LIN {X 0,Y 278.878,Z 465.633,A -85,B 0,C 180,E1 8845.226,E2 8845.226} C_VEL
LIN {X 0,Y 273.338,Z 453.94,A -85,B 0,C 180,E1 8842.303,E2 8842.303} C_VEL
LIN {X 0,Y 267.946,Z 443.512,A -85,B 0,C 180,E1 8839.057,E2 8839.057} C_VEL
LIN {X 0,Y 262.361,Z 433.364,A -85,B 0,C 180,E1 8835.019,E2 8835.019} C_VEL
LIN {X 0,Y 258.426,Z 426.882,A -85,B 0,C 180,E1 8831.493,E2 8831.493} C_VEL
LIN {X 0,Y 256.433,Z 423.717,A -85,B 0,C 180,E1 8829.312,E2 8829.312} C_VEL
LIN {X 0,Y 254.428,Z 420.112,A -85,B 0,C 180,E1 8826.543,E2 8826.543} C_VEL
LIN {X 0,Y 252.019,Z 415.913,A -85,B 0,C 180,E1 8821.364,E2 8821.364} C_VEL
LIN {X 0,Y 251.317,Z 414.93,A -85,B 0,C 180,E1 8815.664,E2 8815.664} C_VEL
LIN {X 0,Y 252.963,Z 416.019,A -85,B 0,C 180,E1 8809.754,E2 8809.754} C_VEL
LIN {X 0,Y 256.776,Z 421.342,A -85,B 0,C 180,E1 8803.95,E2 8803.95} C_VEL
LIN {X 0,Y 260.32,Z 426.562,A -85,B 0,C 180,E1 8800.361,E2 8800.361} C_VEL
LIN {X 0,Y 263.768,Z 431.814,A -85,B 0,C 180,E1 8797.547,E2 8797.547} C_VEL
LIN {X 0,Y 267.986,Z 438.368,A -85,B 0,C 180,E1 8794.65,E2 8794.65} C_VEL
LIN {X 0,Y 273.416,Z 447.764,A -85,B 0,C 180,E1 8791.435,E2 8791.435} C_VEL
LIN {X 0,Y 278.64,Z 457.79,A -85,B 0,C 180,E1 8788.724,E2 8788.724} C_VEL
LIN {X 0,Y 269.524,Z 577.471,A -85,B 0,C 180,E1 8786.054,E2 8786.054} C_VEL
LIN {X 0,Y 267.466,Z 596.812,A -85,B 0,C 180,E1 8785.36,E2 8785.36} C_VEL
LIN {X 0,Y 264.312,Z 615.233,A -85,B 0,C 180,E1 8784.419,E2 8784.419} C_VEL
LIN {X 0,Y 259.903,Z 633.791,A -85,B 0,C 180,E1 8783.145,E2 8783.145} C_VEL
LIN {X 0,Y 254.582,Z 651.308,A -85,B 0,C 180,E1 8781.583,E2 8781.583} C_VEL
LIN {X 0,Y 248.111,Z 668.635,A -85,B 0,C 180,E1 8779.608,E2 8779.608} C_VEL
LIN {X 0,Y 240.971,Z 684.785,A -85,B 0,C 180,E1 8777.257,E2 8777.257} C_VEL
LIN {X 0,Y 233.585,Z 699.288,A -85,B 0,C 180,E1 8774.586,E2 8774.586} C_VEL
LIN {X 0,Y 225.6,Z 713.172,A -85,B 0,C 180,E1 8771.327,E2 8771.327} C_VEL
LIN {X 0,Y 217.777,Z 725.421,A -85,B 0,C 180,E1 8767.634,E2 8767.634} C_VEL
LIN {X 0,Y 210.347,Z 736.116,A -85,B 0,C 180,E1 8763.461,E2 8763.461} C_VEL
LIN {X 0,Y 203.591,Z 745.264,A -85,B 0,C 180,E1 8758.769,E2 8758.769} C_VEL
LIN {X 0,Y 197.74,Z 752.844,A -85,B 0,C 180,E1 8753.544,E2 8753.544} C_VEL
LIN {X 0,Y 193.295,Z 758.557,A -85,B 0,C 180,E1 8748.081,E2 8748.081} C_VEL
LIN {X 0,Y 190.101,Z 762.723,A -85,B 0,C 180,E1 8742.145,E2 8742.145} C_VEL
LIN {X 0,Y 188.303,Z 765.165,A -85,B 0,C 180,E1 8736.096,E2 8736.096} C_VEL
LIN {X 0,Y 187.747,Z 765.976,A -85,B 0,C 180,E1 8730,E2 8730} C_VEL
LIN {X 0,Y 188.29,Z 765.2,A -85,B 0,C 180,E1 8723.904,E2 8723.904} C_VEL
LIN {X 0,Y 190.069,Z 762.799,A -85,B 0,C 180,E1 8717.853,E2 8717.853} C_VEL
LIN {X 0,Y 193.245,Z 758.673,A -85,B 0,C 180,E1 8711.915,E2 8711.915} C_VEL
LIN {X 0,Y 197.948,Z 752.674,A -85,B 0,C 180,E1 8706.167,E2 8706.167} C_VEL
LIN {X 0,Y 203.857,Z 745.036,A -85,B 0,C 180,E1 8700.951,E2 8700.951} C_VEL
LIN {X 0,Y 210.664,Z 735.828,A -85,B 0,C 180,E1 8696.269,E2 8696.269} C_VEL
LIN {X 0,Y 218.141,Z 725.064,A -85,B 0,C 180,E1 8692.108,E2 8692.108} C_VEL
LIN {X 0,Y 226.001,Z 712.736,A -85,B 0,C 180,E1 8688.425,E2 8688.425} C_VEL
LIN {X 0,Y 234.026,Z 698.729,A -85,B 0,C 180,E1 8685.172,E2 8685.172} C_VEL
LIN {X 0,Y 241.439,Z 684.148,A -85,B 0,C 180,E1 8682.513,E2 8682.513} C_VEL
LIN {X 0,Y 248.603,Z 667.849,A -85,B 0,C 180,E1 8680.17,E2 8680.17} C_VEL
LIN {X 0,Y 255.089,Z 650.314,A -85,B 0,C 180,E1 8678.199,E2 8678.199} C_VEL
LIN {X 0,Y 260.429,Z 632.572,A -85,B 0,C 180,E1 8676.641,E2 8676.641} C_VEL
LIN {X 0,Y 264.883,Z 613.37,A -85,B 0,C 180,E1 8675.356,E2 8675.356} C_VEL
LIN {X 0,Y 268.08,Z 593.774,A -85,B 0,C 180,E1 8674.394,E2 8674.394} C_VEL
LIN {X 0,Y 270.011,Z 573.44,A -85,B 0,C 180,E1 8673.717,E2 8673.717} C_VEL
LIN {X 0,Y 278.808,Z 457.69,A -85,B 0,C 180,E1 8671.152,E2 8671.152} C_VEL
LIN {X 0,Y 272.497,Z 445.95,A -85,B 0,C 180,E1 8667.839,E2 8667.839} C_VEL
LIN {X 0,Y 267.272,Z 437.11,A -85,B 0,C 180,E1 8664.653,E2 8664.653} C_VEL
LIN {X 0,Y 262.532,Z 429.641,A -85,B 0,C 180,E1 8661.212,E2 8661.212} C_VEL
LIN {X 0,Y 259.127,Z 424.746,A -85,B 0,C 180,E1 8658.213,E2 8658.213} C_VEL
LIN {X 0,Y 256.354,Z 420.667,A -85,B 0,C 180,E1 8655.149,E2 8655.149} C_VEL
LIN {X 0,Y 253.062,Z 416.095,A -85,B 0,C 180,E1 8649.782,E2 8649.782} C_VEL
LIN {X 0,Y 251.573,Z 415.164,A -85,B 0,C 180,E1 8643.875,E2 8643.875} C_VEL
LIN {X 0,Y 252.355,Z 416.185,A -85,B 0,C 180,E1 8638.411,E2 8638.411} C_VEL
LIN {X 0,Y 255.115,Z 421.076,A -85,B 0,C 180,E1 8632.796,E2 8632.796} C_VEL
LIN {X 0,Y 258.442,Z 426.742,A -85,B 0,C 180,E1 8628.734,E2 8628.734} C_VEL
LIN {X 0,Y 261.024,Z 431.187,A -85,B 0,C 180,E1 8626.272,E2 8626.272} C_VEL
LIN {X 0,Y 262.586,Z 435.115,A -85,B 0,C 180,E1 8624.85,E2 8624.85} C_VEL
LIN {X 0,Y 264.574,Z 443.488,A -85,B 0,C 180,E1 8622.933,E2 8622.933} C_VEL
LIN {X 0,Y 266.814,Z 452.064,A -85,B 0,C 180,E1 8621.05,E2 8621.05} C_VEL
LIN {X 0,Y 267.623,Z 454.063,A -85,B 0,C 180,E1 8620.49,E2 8620.49} C_VEL
LIN {X 0,Y 272.716,Z 464.616,A -85,B 0,C 180,E1 8617.416,E2 8617.416} C_VEL
LIN {X 0,Y 274.98,Z 470.078,A -85,B 0,C 180,E1 8616.14,E2 8616.14} C_VEL
LIN {X 0,Y 262.311,Z 614.422,A -85,B 0,C 180,E1 8612.779,E2 8612.779} C_VEL
LIN {X 0,Y 258.795,Z 635.834,A -85,B 0,C 180,E1 8612.035,E2 8612.035} C_VEL
LIN {X 0,Y 253.894,Z 656.209,A -85,B 0,C 180,E1 8611.07,E2 8611.07} C_VEL
LIN {X 0,Y 247.581,Z 676.274,A -85,B 0,C 180,E1 8609.793,E2 8609.793} C_VEL
LIN {X 0,Y 240.198,Z 695.651,A -85,B 0,C 180,E1 8608.12,E2 8608.12} C_VEL
LIN {X 0,Y 232.104,Z 713.934,A -85,B 0,C 180,E1 8606.019,E2 8606.019} C_VEL
LIN {X 0,Y 223.481,Z 731.176,A -85,B 0,C 180,E1 8603.423,E2 8603.423} C_VEL
LIN {X 0,Y 214.547,Z 747.362,A -85,B 0,C 180,E1 8600.258,E2 8600.258} C_VEL
LIN {X 0,Y 205.621,Z 762.427,A -85,B 0,C 180,E1 8596.428,E2 8596.428} C_VEL
LIN {X 0,Y 197.354,Z 775.9,A -85,B 0,C 180,E1 8591.969,E2 8591.969} C_VEL
LIN {X 0,Y 190.055,Z 787.822,A -85,B 0,C 180,E1 8586.85,E2 8586.85} C_VEL
LIN {X 0,Y 184.137,Z 798.176,A -85,B 0,C 180,E1 8581.053,E2 8581.053} C_VEL
LIN {X 0,Y 180.13,Z 806.495,A -85,B 0,C 180,E1 8574.951,E2 8574.951} C_VEL
LIN {X 0,Y 177.989,Z 812.955,A -85,B 0,C 180,E1 8568.674,E2 8568.674} C_VEL
LIN {X 0,Y 177.55,Z 817.657,A -85,B 0,C 180,E1 8562.356,E2 8562.356} C_VEL
LIN {X 0,Y 178.282,Z 820.523,A -85,B 0,C 180,E1 8556.44,E2 8556.44} C_VEL
LIN {X 0,Y 179.036,Z 821.548,A -85,B 0,C 180,E1 8551.92,E2 8551.92} C_VEL
LIN {X 0,Y 179.07,Z 821.577,A -85,B 0,C 180,E1 8548.4,E2 8548.4} C_VEL
LIN {X 0,Y 178.404,Z 820.702,A -85,B 0,C 180,E1 8544.21,E2 8544.21} C_VEL
LIN {X 0,Y 177.589,Z 818.027,A -85,B 0,C 180,E1 8538.306,E2 8538.306} C_VEL
LIN {X 0,Y 177.869,Z 813.516,A -85,B 0,C 180,E1 8531.991,E2 8531.991} C_VEL
LIN {X 0,Y 179.816,Z 807.245,A -85,B 0,C 180,E1 8525.703,E2 8525.703} C_VEL
LIN {X 0,Y 183.877,Z 798.609,A -85,B 0,C 180,E1 8519.261,E2 8519.261} C_VEL
LIN {X 0,Y 189.692,Z 788.341,A -85,B 0,C 180,E1 8513.445,E2 8513.445} C_VEL
LIN {X 0,Y 196.965,Z 776.407,A -85,B 0,C 180,E1 8508.263,E2 8508.263} C_VEL
LIN {X 0,Y 205.148,Z 763.047,A -85,B 0,C 180,E1 8503.795,E2 8503.795} C_VEL
LIN {X 0,Y 213.949,Z 748.192,A -85,B 0,C 180,E1 8499.968,E2 8499.968} C_VEL
LIN {X 0,Y 222.83,Z 732.143,A -85,B 0,C 180,E1 8496.782,E2 8496.782} C_VEL
LIN {X 0,Y 231.368,Z 715.151,A -85,B 0,C 180,E1 8494.18,E2 8494.18} C_VEL
LIN {X 0,Y 239.105,Z 697.83,A -85,B 0,C 180,E1 8492.138,E2 8492.138} C_VEL
LIN {X 0,Y 246.063,Z 679.96,A -85,B 0,C 180,E1 8490.524,E2 8490.524} C_VEL
LIN {X 0,Y 252.141,Z 661.532,A -85,B 0,C 180,E1 8489.264,E2 8489.264} C_VEL
LIN {X 0,Y 257.488,Z 640.986,A -85,B 0,C 180,E1 8488.212,E2 8488.212} C_VEL
LIN {X 0,Y 261.349,Z 619.931,A -85,B 0,C 180,E1 8487.418,E2 8487.418} C_VEL
LIN {X 0,Y 264.036,Z 594.652,A -85,B 0,C 180,E1 8486.746,E2 8486.746} C_VEL
LIN {X 0,Y 274.757,Z 469.441,A -85,B 0,C 180,E1 8483.824,E2 8483.824} C_VEL
LIN {X 0,Y 269.41,Z 457.799,A -85,B 0,C 180,E1 8480.758,E2 8480.758} C_VEL
LIN {X 0,Y 263.947,Z 447.113,A -85,B 0,C 180,E1 8477.129,E2 8477.129} C_VEL
LIN {X 0,Y 259.778,Z 439.543,A -85,B 0,C 180,E1 8473.805,E2 8473.805} C_VEL
LIN {X 0,Y 256.77,Z 434.226,A -85,B 0,C 180,E1 8470.886,E2 8470.886} C_VEL
LIN {X 0,Y 253.434,Z 428.163,A -85,B 0,C 180,E1 8466.569,E2 8466.569} C_VEL
LIN {X 0,Y 250.96,Z 423.8,A -85,B 0,C 180,E1 8461.141,E2 8461.141} C_VEL
LIN {X 0,Y 250.345,Z 422.871,A -85,B 0,C 180,E1 8455.647,E2 8455.647} C_VEL
LIN {X 0,Y 252.001,Z 423.991,A -85,B 0,C 180,E1 8449.714,E2 8449.714} C_VEL
LIN {X 0,Y 255.526,Z 429.237,A -85,B 0,C 180,E1 8444.219,E2 8444.219} C_VEL
LIN {X 0,Y 258.761,Z 434.142,A -85,B 0,C 180,E1 8440.825,E2 8440.825} C_VEL
LIN {X 0,Y 262.133,Z 439.449,A -85,B 0,C 180,E1 8437.971,E2 8437.971} C_VEL
LIN {X 0,Y 266.367,Z 446.383,A -85,B 0,C 180,E1 8434.961,E2 8434.961} C_VEL
LIN {X 0,Y 271.172,Z 455.032,A -85,B 0,C 180,E1 8432.017,E2 8432.017} C_VEL
LIN {X 0,Y 274.625,Z 461.918,A -85,B 0,C 180,E1 8430.11,E2 8430.11} C_VEL
LIN {X 0,Y 265.44,Z 578.24,A -85,B 0,C 180,E1 8427.518,E2 8427.518} C_VEL
LIN {X 0,Y 263.304,Z 597.581,A -85,B 0,C 180,E1 8426.825,E2 8426.825} C_VEL
LIN {X 0,Y 260.034,Z 616.06,A -85,B 0,C 180,E1 8425.886,E2 8425.886} C_VEL
LIN {X 0,Y 255.561,Z 634.361,A -85,B 0,C 180,E1 8424.639,E2 8424.639} C_VEL
LIN {X 0,Y 250.09,Z 651.862,A -85,B 0,C 180,E1 8423.09,E2 8423.09} C_VEL
LIN {X 0,Y 243.394,Z 669.282,A -85,B 0,C 180,E1 8421.118,E2 8421.118} C_VEL
LIN {X 0,Y 235.981,Z 685.526,A -85,B 0,C 180,E1 8418.762,E2 8418.762} C_VEL
LIN {X 0,Y 228.025,Z 700.565,A -85,B 0,C 180,E1 8415.98,E2 8415.98} C_VEL
LIN {X 0,Y 219.721,Z 714.42,A -85,B 0,C 180,E1 8412.689,E2 8412.689} C_VEL
LIN {X 0,Y 211.561,Z 726.652,A -85,B 0,C 180,E1 8408.944,E2 8408.944} C_VEL
LIN {X 0,Y 203.781,Z 737.336,A -85,B 0,C 180,E1 8404.69,E2 8404.69} C_VEL
LIN {X 0,Y 196.675,Z 746.477,A -85,B 0,C 180,E1 8399.881,E2 8399.881} C_VEL
LIN {X 0,Y 190.493,Z 754.053,A -85,B 0,C 180,E1 8394.497,E2 8394.497} C_VEL
LIN {X 0,Y 185.77,Z 759.763,A -85,B 0,C 180,E1 8388.84,E2 8388.84} C_VEL
LIN {X 0,Y 182.363,Z 763.927,A -85,B 0,C 180,E1 8382.668,E2 8382.668} C_VEL
LIN {X 0,Y 180.435,Z 766.367,A -85,B 0,C 180,E1 8376.363,E2 8376.363} C_VEL
LIN {X 0,Y 179.838,Z 767.178,A -85,B 0,C 180,E1 8370,E2 8370} C_VEL
LIN {X 0,Y 180.422,Z 766.402,A -85,B 0,C 180,E1 8363.637,E2 8363.637} C_VEL
LIN {X 0,Y 182.33,Z 764.002,A -85,B 0,C 180,E1 8357.329,E2 8357.329} C_VEL
LIN {X 0,Y 185.719,Z 759.877,A -85,B 0,C 180,E1 8351.155,E2 8351.155} C_VEL
LIN {X 0,Y 190.717,Z 753.881,A -85,B 0,C 180,E1 8345.203,E2 8345.203} C_VEL
LIN {X 0,Y 196.958,Z 746.25,A -85,B 0,C 180,E1 8339.831,E2 8339.831} C_VEL
LIN {X 0,Y 204.119,Z 737.048,A -85,B 0,C 180,E1 8335.034,E2 8335.034} C_VEL
LIN {X 0,Y 211.947,Z 726.296,A -85,B 0,C 180,E1 8330.793,E2 8330.793} C_VEL
LIN {X 0,Y 220.146,Z 713.986,A -85,B 0,C 180,E1 8327.059,E2 8327.059} C_VEL
LIN {X 0,Y 228.485,Z 700.025,A -85,B 0,C 180,E1 8323.778,E2 8323.778} C_VEL
LIN {X 0,Y 236.481,Z 684.837,A -85,B 0,C 180,E1 8321.002,E2 8321.002} C_VEL
LIN {X 0,Y 243.906,Z 668.454,A -85,B 0,C 180,E1 8318.657,E2 8318.657} C_VEL
LIN {X 0,Y 250.266,Z 651.876,A -85,B 0,C 180,E1 8316.793,E2 8316.793} C_VEL
LIN {X 0,Y 255.814,Z 634.148,A -85,B 0,C 180,E1 8315.228,E2 8315.228} C_VEL
LIN {X 0,Y 260.374,Z 615.388,A -85,B 0,C 180,E1 8313.96,E2 8313.96} C_VEL
LIN {X 0,Y 263.777,Z 595.743,A -85,B 0,C 180,E1 8312.979,E2 8312.979} C_VEL
LIN {X 0,Y 265.852,Z 575.618,A -85,B 0,C 180,E1 8312.291,E2 8312.291} C_VEL
LIN {X 0,Y 274.724,Z 461.747,A -85,B 0,C 180,E1 8309.729,E2 8309.729} C_VEL
LIN {X 0,Y 269.186,Z 451.135,A -85,B 0,C 180,E1 8306.589,E2 8306.589} C_VEL
LIN {X 0,Y 264.409,Z 442.959,A -85,B 0,C 180,E1 8303.454,E2 8303.454} C_VEL
LIN {X 0,Y 260.148,Z 436.17,A -85,B 0,C 180,E1 8300.12,E2 8300.12} C_VEL
LIN {X 0,Y 257.621,Z 432.313,A -85,B 0,C 180,E1 8297.739,E2 8297.739} C_VEL
LIN {X 0,Y 255.045,Z 428.396,A -85,B 0,C 180,E1 8294.763,E2 8294.763} C_VEL
LIN {X 0,Y 252.008,Z 423.989,A -85,B 0,C 180,E1 8289.593,E2 8289.593} C_VEL
LIN {X 0,Y 250.592,Z 423.106,A -85,B 0,C 180,E1 8283.661,E2 8283.661} C_VEL
LIN {X 0,Y 251.362,Z 424.279,A -85,B 0,C 180,E1 8278.405,E2 8278.405} C_VEL
LIN {X 0,Y 253.873,Z 428.918,A -85,B 0,C 180,E1 8273.101,E2 8273.101} C_VEL
LIN {X 0,Y 256.901,Z 434.265,A -85,B 0,C 180,E1 8269.233,E2 8269.233} C_VEL
LIN {X 0,Y 260.684,Z 440.814,A -85,B 0,C 180,E1 8265.621,E2 8265.621} C_VEL
LIN {X 0,Y 265.967,Z 450.804,A -85,B 0,C 180,E1 8261.592,E2 8261.592} C_VEL
LIN {X 0,Y 267.623,Z 454.063,A -85,B 0,C 180,E1 8260.49,E2 8260.49} C_VEL
LIN {X 0,Y 268.653,Z 457.702,A -85,B 0,C 180,E1 8259.728,E2 8259.728} C_VEL
LIN {X 0,Y 270.267,Z 470.787,A -85,B 0,C 180,E1 8258.119,E2 8258.119} C_VEL
LIN {X 0,Y 271.051,Z 473.538,A -85,B 0,C 180,E1 8257.597,E2 8257.597} C_VEL
LIN {X 0,Y 258.457,Z 613.492,A -85,B 0,C 180,E1 8254.336,E2 8254.336} C_VEL
LIN {X 0,Y 254.871,Z 634.831,A -85,B 0,C 180,E1 8253.607,E2 8253.607} C_VEL
LIN {X 0,Y 249.872,Z 655.168,A -85,B 0,C 180,E1 8252.661,E2 8252.661} C_VEL
LIN {X 0,Y 243.592,Z 674.701,A -85,B 0,C 180,E1 8251.446,E2 8251.446} C_VEL
LIN {X 0,Y 235.986,Z 694.185,A -85,B 0,C 180,E1 8249.804,E2 8249.804} C_VEL
LIN {X 0,Y 227.614,Z 712.526,A -85,B 0,C 180,E1 8247.735,E2 8247.735} C_VEL
LIN {X 0,Y 218.527,Z 730.074,A -85,B 0,C 180,E1 8245.116,E2 8245.116} C_VEL
LIN {X 0,Y 209.154,Z 746.368,A -85,B 0,C 180,E1 8241.926,E2 8241.926} C_VEL
LIN {X 0,Y 199.978,Z 761.113,A -85,B 0,C 180,E1 8238.155,E2 8238.155} C_VEL
LIN {X 0,Y 191.242,Z 774.603,A -85,B 0,C 180,E1 8233.639,E2 8233.639} C_VEL
LIN {X 0,Y 183.44,Z 786.534,A -85,B 0,C 180,E1 8228.415,E2 8228.415} C_VEL
LIN {X 0,Y 177.041,Z 796.897,A -85,B 0,C 180,E1 8222.446,E2 8222.446} C_VEL
LIN {X 0,Y 172.62,Z 805.225,A -85,B 0,C 180,E1 8216.116,E2 8216.116} C_VEL
LIN {X 0,Y 170.181,Z 811.698,A -85,B 0,C 180,E1 8209.565,E2 8209.565} C_VEL
LIN {X 0,Y 169.577,Z 816.415,A -85,B 0,C 180,E1 8202.947,E2 8202.947} C_VEL
LIN {X 0,Y 170.287,Z 819.301,A -85,B 0,C 180,E1 8196.744,E2 8196.744} C_VEL
LIN {X 0,Y 171.107,Z 820.343,A -85,B 0,C 180,E1 8192.009,E2 8192.009} C_VEL
LIN {X 0,Y 171.178,Z 820.405,A -85,B 0,C 180,E1 8188.661,E2 8188.661} C_VEL
LIN {X 0,Y 170.476,Z 819.577,A -85,B 0,C 180,E1 8184.278,E2 8184.278} C_VEL
LIN {X 0,Y 169.621,Z 816.985,A -85,B 0,C 180,E1 8178.094,E2 8178.094} C_VEL
LIN {X 0,Y 169.97,Z 812.559,A -85,B 0,C 180,E1 8171.479,E2 8171.479} C_VEL
LIN {X 0,Y 172.273,Z 805.975,A -85,B 0,C 180,E1 8164.566,E2 8164.566} C_VEL
LIN {X 0,Y 176.757,Z 797.329,A -85,B 0,C 180,E1 8157.879,E2 8157.879} C_VEL
LIN {X 0,Y 183.113,Z 786.955,A -85,B 0,C 180,E1 8151.839,E2 8151.839} C_VEL
LIN {X 0,Y 190.759,Z 775.213,A -85,B 0,C 180,E1 8146.637,E2 8146.637} C_VEL
LIN {X 0,Y 199.421,Z 761.827,A -85,B 0,C 180,E1 8142.096,E2 8142.096} C_VEL
LIN {X 0,Y 208.727,Z 746.868,A -85,B 0,C 180,E1 8138.225,E2 8138.225} C_VEL
LIN {X 0,Y 217.99,Z 730.79,A -85,B 0,C 180,E1 8135.045,E2 8135.045} C_VEL
LIN {X 0,Y 226.895,Z 713.67,A -85,B 0,C 180,E1 8132.45,E2 8132.45} C_VEL
LIN {X 0,Y 235.227,Z 695.538,A -85,B 0,C 180,E1 8130.362,E2 8130.362} C_VEL
LIN {X 0,Y 242.416,Z 677.385,A -85,B 0,C 180,E1 8128.784,E2 8128.784} C_VEL
LIN {X 0,Y 248.711,Z 658.403,A -85,B 0,C 180,E1 8127.548,E2 8127.548} C_VEL
LIN {X 0,Y 253.921,Z 638.253,A -85,B 0,C 180,E1 8126.563,E2 8126.563} C_VEL
LIN {X 0,Y 257.673,Z 617.588,A -85,B 0,C 180,E1 8125.814,E2 8125.814} C_VEL
LIN {X 0,Y 260.622,Z 589.211,A -85,B 0,C 180,E1 8125.086,E2 8125.086} C_VEL
LIN {X 0,Y 270.847,Z 473.338,A -85,B 0,C 180,E1 8122.405,E2 8122.405} C_VEL
LIN {X 0,Y 266.038,Z 462.77,A -85,B 0,C 180,E1 8119.427,E2 8119.427} C_VEL
LIN {X 0,Y 261.467,Z 453.484,A -85,B 0,C 180,E1 8116.152,E2 8116.152} C_VEL
LIN {X 0,Y 257.896,Z 446.68,A -85,B 0,C 180,E1 8113.109,E2 8113.109} C_VEL
LIN {X 0,Y 254.958,Z 441.205,A -85,B 0,C 180,E1 8110.05,E2 8110.05} C_VEL
LIN {X 0,Y 251.865,Z 435.512,A -85,B 0,C 180,E1 8105.695,E2 8105.695} C_VEL
LIN {X 0,Y 249.905,Z 431.687,A -85,B 0,C 180,E1 8100.917,E2 8100.917} C_VEL
LIN {X 0,Y 249.389,Z 430.818,A -85,B 0,C 180,E1 8095.4,E2 8095.4} C_VEL
LIN {X 0,Y 250.937,Z 431.891,A -85,B 0,C 180,E1 8089.902,E2 8089.902} C_VEL
LIN {X 0,Y 254.192,Z 436.961,A -85,B 0,C 180,E1 8084.602,E2 8084.602} C_VEL
LIN {X 0,Y 257.218,Z 441.719,A -85,B 0,C 180,E1 8081.295,E2 8081.295} C_VEL
LIN {X 0,Y 260.737,Z 447.429,A -85,B 0,C 180,E1 8078.221,E2 8078.221} C_VEL
LIN {X 0,Y 265.223,Z 455.175,A -85,B 0,C 180,E1 8074.965,E2 8074.965} C_VEL
LIN {X 0,Y 270.149,Z 464.689,A -85,B 0,C 180,E1 8071.902,E2 8071.902} C_VEL
LIN {X 0,Y 270.764,Z 466.184,A -85,B 0,C 180,E1 8071.534,E2 8071.534} C_VEL
LIN {X 0,Y 261.543,Z 578.894,A -85,B 0,C 180,E1 8069.031,E2 8069.031} C_VEL
LIN {X 0,Y 259.335,Z 598.253,A -85,B 0,C 180,E1 8068.341,E2 8068.341} C_VEL
LIN {X 0,Y 256.033,Z 616.456,A -85,B 0,C 180,E1 8067.426,E2 8067.426} C_VEL
LIN {X 0,Y 251.465,Z 634.7,A -85,B 0,C 180,E1 8066.2,E2 8066.2} C_VEL
LIN {X 0,Y 245.442,Z 653.314,A -85,B 0,C 180,E1 8064.559,E2 8064.559} C_VEL
LIN {X 0,Y 238.524,Z 670.647,A -85,B 0,C 180,E1 8062.592,E2 8062.592} C_VEL
LIN {X 0,Y 230.865,Z 686.815,A -85,B 0,C 180,E1 8060.239,E2 8060.239} C_VEL
LIN {X 0,Y 222.606,Z 701.837,A -85,B 0,C 180,E1 8057.443,E2 8057.443} C_VEL
LIN {X 0,Y 213.973,Z 715.667,A -85,B 0,C 180,E1 8054.125,E2 8054.125} C_VEL
LIN {X 0,Y 205.461,Z 727.883,A -85,B 0,C 180,E1 8050.332,E2 8050.332} C_VEL
LIN {X 0,Y 197.315,Z 738.556,A -85,B 0,C 180,E1 8046.001,E2 8046.001} C_VEL
LIN {X 0,Y 189.838,Z 747.69,A -85,B 0,C 180,E1 8041.074,E2 8041.074} C_VEL
LIN {X 0,Y 183.302,Z 755.261,A -85,B 0,C 180,E1 8035.525,E2 8035.525} C_VEL
LIN {X 0,Y 178.101,Z 761.156,A -85,B 0,C 180,E1 8029.41,E2 8029.41} C_VEL
LIN {X 0,Y 174.64,Z 765.131,A -85,B 0,C 180,E1 8023.239,E2 8023.239} C_VEL
LIN {X 0,Y 172.572,Z 767.569,A -85,B 0,C 180,E1 8016.654,E2 8016.654} C_VEL
LIN {X 0,Y 171.929,Z 768.379,A -85,B 0,C 180,E1 8010,E2 8010} C_VEL
LIN {X 0,Y 172.558,Z 767.603,A -85,B 0,C 180,E1 8003.345,E2 8003.345} C_VEL
LIN {X 0,Y 174.606,Z 765.204,A -85,B 0,C 180,E1 7996.759,E2 7996.759} C_VEL
LIN {X 0,Y 178.23,Z 761.081,A -85,B 0,C 180,E1 7990.331,E2 7990.331} C_VEL
LIN {X 0,Y 183.543,Z 755.089,A -85,B 0,C 180,E1 7984.165,E2 7984.165} C_VEL
LIN {X 0,Y 190.141,Z 747.462,A -85,B 0,C 180,E1 7978.629,E2 7978.629} C_VEL
LIN {X 0,Y 197.674,Z 738.268,A -85,B 0,C 180,E1 7973.716,E2 7973.716} C_VEL
LIN {X 0,Y 205.871,Z 727.526,A -85,B 0,C 180,E1 7969.4,E2 7969.4} C_VEL
LIN {X 0,Y 214.422,Z 715.233,A -85,B 0,C 180,E1 7965.618,E2 7965.618} C_VEL
LIN {X 0,Y 223.091,Z 701.302,A -85,B 0,C 180,E1 7962.313,E2 7962.313} C_VEL
LIN {X 0,Y 231.381,Z 686.158,A -85,B 0,C 180,E1 7959.527,E2 7959.527} C_VEL
LIN {X 0,Y 239.064,Z 669.839,A -85,B 0,C 180,E1 7957.182,E2 7957.182} C_VEL
LIN {X 0,Y 245.998,Z 652.299,A -85,B 0,C 180,E1 7955.22,E2 7955.22} C_VEL
LIN {X 0,Y 251.698,Z 634.574,A -85,B 0,C 180,E1 7953.674,E2 7953.674} C_VEL
LIN {X 0,Y 256.472,Z 615.362,A -85,B 0,C 180,E1 7952.396,E2 7952.396} C_VEL
LIN {X 0,Y 259.942,Z 595.562,A -85,B 0,C 180,E1 7951.429,E2 7951.429} C_VEL
LIN {X 0,Y 262.042,Z 575.24,A -85,B 0,C 180,E1 7950.751,E2 7950.751} C_VEL
LIN {X 0,Y 270.904,Z 465.97,A -85,B 0,C 180,E1 7948.313,E2 7948.313} C_VEL
LIN {X 0,Y 265.845,Z 456.132,A -85,B 0,C 180,E1 7945.211,E2 7945.211} C_VEL
LIN {X 0,Y 261.321,Z 448.177,A -85,B 0,C 180,E1 7941.964,E2 7941.964} C_VEL
LIN {X 0,Y 257.639,Z 442.271,A -85,B 0,C 180,E1 7938.791,E2 7938.791} C_VEL
LIN {X 0,Y 255.622,Z 439.169,A -85,B 0,C 180,E1 7936.708,E2 7936.708} C_VEL
LIN {X 0,Y 253.747,Z 436.123,A -85,B 0,C 180,E1 7934.374,E2 7934.374} C_VEL
LIN {X 0,Y 250.952,Z 431.883,A -85,B 0,C 180,E1 7929.402,E2 7929.402} C_VEL
LIN {X 0,Y 249.613,Z 431.063,A -85,B 0,C 180,E1 7923.445,E2 7923.445} C_VEL
LIN {X 0,Y 250.31,Z 432.173,A -85,B 0,C 180,E1 7918.627,E2 7918.627} C_VEL
LIN {X 0,Y 252.595,Z 436.657,A -85,B 0,C 180,E1 7913.482,E2 7913.482} C_VEL
LIN {X 0,Y 255.473,Z 441.965,A -85,B 0,C 180,E1 7909.629,E2 7909.629} C_VEL
LIN {X 0,Y 259.181,Z 448.801,A -85,B 0,C 180,E1 7905.934,E2 7905.934} C_VEL
LIN {X 0,Y 263.838,Z 457.95,A -85,B 0,C 180,E1 7902.238,E2 7902.238} C_VEL
LIN {X 0,Y 268.608,Z 468.029,A -85,B 0,C 180,E1 7899.063,E2 7899.063} C_VEL
LIN {X 0,Y 271.051,Z 473.538,A -85,B 0,C 180,E1 7897.597,E2 7897.597} C_VEL
LIN {X 0,Y 271.539,Z 476.413,A -85,B 0,C 180,E1 7897.208,E2 7897.208} C_VEL
LIN {X 0,Y 271.269,Z 480.92,A -85,B 0,C 180,E1 7897.051,E2 7897.051} C_VEL
LIN {X 0,Y 269.929,Z 487.325,A -85,B 0,C 180,E1 7897.239,E2 7897.239} C_VEL
LIN {X 0,Y 265.57,Z 502.194,A -85,B 0,C 180,E1 7898.257,E2 7898.257} C_VEL
LIN {X 0,Y 264.534,Z 508.324,A -85,B 0,C 180,E1 7898.34,E2 7898.34} C_VEL
LIN {X 0,Y 254.757,Z 612.84,A -85,B 0,C 180,E1 7895.931,E2 7895.931} C_VEL
LIN {X 0,Y 251.088,Z 634.078,A -85,B 0,C 180,E1 7895.216,E2 7895.216} C_VEL
LIN {X 0,Y 245.844,Z 654.788,A -85,B 0,C 180,E1 7894.266,E2 7894.266} C_VEL
LIN {X 0,Y 239.415,Z 674.224,A -85,B 0,C 180,E1 7893.075,E2 7893.075} C_VEL
LIN {X 0,Y 231.603,Z 693.598,A -85,B 0,C 180,E1 7891.463,E2 7891.463} C_VEL
LIN {X 0,Y 222.975,Z 711.859,A -85,B 0,C 180,E1 7889.422,E2 7889.422} C_VEL
LIN {X 0,Y 213.717,Z 729.073,A -85,B 0,C 180,E1 7886.868,E2 7886.868} C_VEL
LIN {X 0,Y 204.038,Z 745.225,A -85,B 0,C 180,E1 7883.715,E2 7883.715} C_VEL
LIN {X 0,Y 194.533,Z 759.801,A -85,B 0,C 180,E1 7879.979,E2 7879.979} C_VEL
LIN {X 0,Y 185.3,Z 773.305,A -85,B 0,C 180,E1 7875.417,E2 7875.417} C_VEL
LIN {X 0,Y 176.976,Z 785.247,A -85,B 0,C 180,E1 7870.094,E2 7870.094} C_VEL
LIN {X 0,Y 170.06,Z 795.62,A -85,B 0,C 180,E1 7863.954,E2 7863.954} C_VEL
LIN {X 0,Y 165.185,Z 803.954,A -85,B 0,C 180,E1 7857.388,E2 7857.388} C_VEL
LIN {X 0,Y 162.407,Z 810.439,A -85,B 0,C 180,E1 7850.543,E2 7850.543} C_VEL
LIN {X 0,Y 161.613,Z 815.173,A -85,B 0,C 180,E1 7843.597,E2 7843.597} C_VEL
LIN {X 0,Y 162.282,Z 818.076,A -85,B 0,C 180,E1 7837.078,E2 7837.078} C_VEL
LIN {X 0,Y 163.175,Z 819.137,A -85,B 0,C 180,E1 7832.107,E2 7832.107} C_VEL
LIN {X 0,Y 163.256,Z 819.202,A -85,B 0,C 180,E1 7828.596,E2 7828.596} C_VEL
LIN {X 0,Y 162.481,Z 818.356,A -85,B 0,C 180,E1 7823.995,E2 7823.995} C_VEL
LIN {X 0,Y 161.638,Z 815.742,A -85,B 0,C 180,E1 7817.497,E2 7817.497} C_VEL
LIN {X 0,Y 162.159,Z 811.3,A -85,B 0,C 180,E1 7810.552,E2 7810.552} C_VEL
LIN {X 0,Y 164.796,Z 804.703,A -85,B 0,C 180,E1 7803.323,E2 7803.323} C_VEL
LIN {X 0,Y 169.748,Z 796.048,A -85,B 0,C 180,E1 7796.381,E2 7796.381} C_VEL
LIN {X 0,Y 176.556,Z 785.763,A -85,B 0,C 180,E1 7790.215,E2 7790.215} C_VEL
LIN {X 0,Y 184.79,Z 773.917,A -85,B 0,C 180,E1 7784.863,E2 7784.863} C_VEL
LIN {X 0,Y 193.946,Z 760.519,A -85,B 0,C 180,E1 7780.273,E2 7780.273} C_VEL
LIN {X 0,Y 203.708,Z 745.539,A -85,B 0,C 180,E1 7776.396,E2 7776.396} C_VEL
LIN {X 0,Y 213.209,Z 729.692,A -85,B 0,C 180,E1 7773.276,E2 7773.276} C_VEL
LIN {X 0,Y 222.597,Z 712.279,A -85,B 0,C 180,E1 7770.666,E2 7770.666} C_VEL
LIN {X 0,Y 231.206,Z 694.085,A -85,B 0,C 180,E1 7768.615,E2 7768.615} C_VEL
LIN {X 0,Y 238.607,Z 675.837,A -85,B 0,C 180,E1 7767.072,E2 7767.072} C_VEL
LIN {X 0,Y 245.023,Z 656.831,A -85,B 0,C 180,E1 7765.873,E2 7765.873} C_VEL
LIN {X 0,Y 250.242,Z 636.931,A -85,B 0,C 180,E1 7764.927,E2 7764.927} C_VEL
LIN {X 0,Y 254.035,Z 616.367,A -85,B 0,C 180,E1 7764.2,E2 7764.2} C_VEL
LIN {X 0,Y 257.092,Z 587.514,A -85,B 0,C 180,E1 7763.472,E2 7763.472} C_VEL
LIN {X 0,Y 267.095,Z 477.349,A -85,B 0,C 180,E1 7760.946,E2 7760.946} C_VEL
LIN {X 0,Y 262.464,Z 466.849,A -85,B 0,C 180,E1 7757.801,E2 7757.801} C_VEL
LIN {X 0,Y 257.967,Z 457.509,A -85,B 0,C 180,E1 7754.19,E2 7754.19} C_VEL
LIN {X 0,Y 254.309,Z 450.317,A -85,B 0,C 180,E1 7750.534,E2 7750.534} C_VEL
LIN {X 0,Y 252.182,Z 446.451,A -85,B 0,C 180,E1 7747.861,E2 7747.861} C_VEL
LIN {X 0,Y 250.603,Z 443.213,A -85,B 0,C 180,E1 7745.265,E2 7745.265} C_VEL
LIN {X 0,Y 248.856,Z 439.575,A -85,B 0,C 180,E1 7740.69,E2 7740.69} C_VEL
LIN {X 0,Y 248.41,Z 438.758,A -85,B 0,C 180,E1 7735.382,E2 7735.382} C_VEL
LIN {X 0,Y 249.865,Z 439.829,A -85,B 0,C 180,E1 7730.091,E2 7730.091} C_VEL
LIN {X 0,Y 252.865,Z 444.683,A -85,B 0,C 180,E1 7724.989,E2 7724.989} C_VEL
LIN {X 0,Y 255.69,Z 449.295,A -85,B 0,C 180,E1 7721.769,E2 7721.769} C_VEL
LIN {X 0,Y 259.434,Z 455.525,A -85,B 0,C 180,E1 7718.404,E2 7718.404} C_VEL
LIN {X 0,Y 264.142,Z 464.247,A -85,B 0,C 180,E1 7714.915,E2 7714.915} C_VEL
LIN {X 0,Y 267.074,Z 470.47,A -85,B 0,C 180,E1 7712.997,E2 7712.997} C_VEL
LIN {X 0,Y 257.843,Z 579.44,A -85,B 0,C 180,E1 7710.592,E2 7710.592} C_VEL
LIN {X 0,Y 255.589,Z 598.711,A -85,B 0,C 180,E1 7709.912,E2 7709.912} C_VEL
LIN {X 0,Y 252.035,Z 617.628,A -85,B 0,C 180,E1 7708.968,E2 7708.968} C_VEL
LIN {X 0,Y 247.178,Z 636.274,A -85,B 0,C 180,E1 7707.715,E2 7707.715} C_VEL
LIN {X 0,Y 241.308,Z 653.871,A -85,B 0,C 180,E1 7706.175,E2 7706.175} C_VEL
LIN {X 0,Y 234.158,Z 671.292,A -85,B 0,C 180,E1 7704.221,E2 7704.221} C_VEL
LIN {X 0,Y 226.228,Z 687.532,A -85,B 0,C 180,E1 7701.877,E2 7701.877} C_VEL
LIN {X 0,Y 217.745,Z 702.468,A -85,B 0,C 180,E1 7699.116,E2 7699.116} C_VEL
LIN {X 0,Y 208.949,Z 716.095,A -85,B 0,C 180,E1 7695.869,E2 7695.869} C_VEL
LIN {X 0,Y 200.025,Z 728.437,A -85,B 0,C 180,E1 7692.052,E2 7692.052} C_VEL
LIN {X 0,Y 191.434,Z 739.221,A -85,B 0,C 180,E1 7687.667,E2 7687.667} C_VEL
LIN {X 0,Y 183.495,Z 748.46,A -85,B 0,C 180,E1 7682.645,E2 7682.645} C_VEL
LIN {X 0,Y 176.504,Z 756.135,A -85,B 0,C 180,E1 7676.947,E2 7676.947} C_VEL
LIN {X 0,Y 170.775,Z 762.231,A -85,B 0,C 180,E1 7670.481,E2 7670.481} C_VEL
LIN {X 0,Y 166.936,Z 766.334,A -85,B 0,C 180,E1 7663.861,E2 7663.861} C_VEL
LIN {X 0,Y 164.713,Z 768.772,A -85,B 0,C 180,E1 7656.973,E2 7656.973} C_VEL
LIN {X 0,Y 164.019,Z 769.581,A -85,B 0,C 180,E1 7650,E2 7650} C_VEL
LIN {X 0,Y 164.698,Z 768.805,A -85,B 0,C 180,E1 7643.026,E2 7643.026} C_VEL
LIN {X 0,Y 167.009,Z 766.307,A -85,B 0,C 180,E1 7635.902,E2 7635.902} C_VEL
LIN {X 0,Y 171.022,Z 762.045,A -85,B 0,C 180,E1 7629.107,E2 7629.107} C_VEL
LIN {X 0,Y 176.764,Z 755.939,A -85,B 0,C 180,E1 7622.732,E2 7622.732} C_VEL
LIN {X 0,Y 183.818,Z 748.206,A -85,B 0,C 180,E1 7617.049,E2 7617.049} C_VEL
LIN {X 0,Y 191.816,Z 738.903,A -85,B 0,C 180,E1 7612.043,E2 7612.043} C_VEL
LIN {X 0,Y 200.458,Z 728.045,A -85,B 0,C 180,E1 7607.674,E2 7607.674} C_VEL
LIN {X 0,Y 209.421,Z 715.62,A -85,B 0,C 180,E1 7603.87,E2 7603.87} C_VEL
LIN {X 0,Y 218.16,Z 702.06,A -85,B 0,C 180,E1 7600.669,E2 7600.669} C_VEL
LIN {X 0,Y 226.765,Z 686.843,A -85,B 0,C 180,E1 7597.887,E2 7597.887} C_VEL
LIN {X 0,Y 234.719,Z 670.442,A -85,B 0,C 180,E1 7595.551,E2 7595.551} C_VEL
LIN {X 0,Y 241.595,Z 653.631,A -85,B 0,C 180,E1 7593.682,E2 7593.682} C_VEL
LIN {X 0,Y 247.56,Z 635.707,A -85,B 0,C 180,E1 7592.124,E2 7592.124} C_VEL
LIN {X 0,Y 252.462,Z 616.691,A -85,B 0,C 180,E1 7590.863,E2 7590.863} C_VEL
LIN {X 0,Y 256.095,Z 596.836,A -85,B 0,C 180,E1 7589.893,E2 7589.893} C_VEL
LIN {X 0,Y 258.309,Z 576.478,A -85,B 0,C 180,E1 7589.21,E2 7589.21} C_VEL
LIN {X 0,Y 267.24,Z 470.279,A -85,B 0,C 180,E1 7586.858,E2 7586.858} C_VEL
LIN {X 0,Y 262.656,Z 461.236,A -85,B 0,C 180,E1 7583.799,E2 7583.799} C_VEL
LIN {X 0,Y 258.568,Z 454.007,A -85,B 0,C 180,E1 7580.603,E2 7580.603} C_VEL
LIN {X 0,Y 255.072,Z 447.992,A -85,B 0,C 180,E1 7577.215,E2 7577.215} C_VEL
LIN {X 0,Y 252.461,Z 443.849,A -85,B 0,C 180,E1 7573.981,E2 7573.981} C_VEL
LIN {X 0,Y 249.889,Z 439.776,A -85,B 0,C 180,E1 7569.21,E2 7569.21} C_VEL
LIN {X 0,Y 248.64,Z 439.004,A -85,B 0,C 180,E1 7563.459,E2 7563.459} C_VEL
LIN {X 0,Y 249.26,Z 440.065,A -85,B 0,C 180,E1 7558.851,E2 7558.851} C_VEL
LIN {X 0,Y 251.292,Z 444.281,A -85,B 0,C 180,E1 7553.948,E2 7553.948} C_VEL
LIN {X 0,Y 254.152,Z 449.837,A -85,B 0,C 180,E1 7549.918,E2 7549.918} C_VEL
LIN {X 0,Y 257.809,Z 457,A -85,B 0,C 180,E1 7546.144,E2 7546.144} C_VEL
LIN {X 0,Y 261.951,Z 465.547,A -85,B 0,C 180,E1 7542.737,E2 7542.737} C_VEL
LIN {X 0,Y 266.413,Z 475.424,A -85,B 0,C 180,E1 7539.63,E2 7539.63} C_VEL
LIN {X 0,Y 267.328,Z 478.005,A -85,B 0,C 180,E1 7539.015,E2 7539.015} C_VEL
LIN {X 0,Y 264.534,Z 508.324,A -85,B 0,C 180,E1 7538.34,E2 7538.34} C_VEL
LIN {X 0,Y 263.392,Z 516.006,A -85,B 0,C 180,E1 7538.372,E2 7538.372} C_VEL
LIN {X 0,Y 258.909,Z 536.454,A -85,B 0,C 180,E1 7539.164,E2 7539.164} C_VEL
LIN {X 0,Y 257.975,Z 543.047,A -85,B 0,C 180,E1 7539.173,E2 7539.173} C_VEL
LIN {X 0,Y 251.242,Z 612.308,A -85,B 0,C 180,E1 7537.568,E2 7537.568} C_VEL
LIN {X 0,Y 247.509,Z 633.326,A -85,B 0,C 180,E1 7536.872,E2 7536.872} C_VEL
LIN {X 0,Y 242.43,Z 653.082,A -85,B 0,C 180,E1 7535.995,E2 7535.995} C_VEL
LIN {X 0,Y 235.832,Z 672.692,A -85,B 0,C 180,E1 7534.833,E2 7534.833} C_VEL
LIN {X 0,Y 227.817,Z 692.134,A -85,B 0,C 180,E1 7533.266,E2 7533.266} C_VEL
LIN {X 0,Y 218.916,Z 710.457,A -85,B 0,C 180,E1 7531.27,E2 7531.27} C_VEL
LIN {X 0,Y 209.325,Z 727.712,A -85,B 0,C 180,E1 7528.758,E2 7528.758} C_VEL
LIN {X 0,Y 199.25,Z 743.894,A -85,B 0,C 180,E1 7525.635,E2 7525.635} C_VEL
LIN {X 0,Y 188.906,Z 759.069,A -85,B 0,C 180,E1 7521.738,E2 7521.738} C_VEL
LIN {X 0,Y 179.014,Z 772.753,A -85,B 0,C 180,E1 7517.026,E2 7517.026} C_VEL
LIN {X 0,Y 170.232,Z 784.585,A -85,B 0,C 180,E1 7511.581,E2 7511.581} C_VEL
LIN {X 0,Y 162.869,Z 794.852,A -85,B 0,C 180,E1 7505.244,E2 7505.244} C_VEL
LIN {X 0,Y 157.364,Z 803.559,A -85,B 0,C 180,E1 7497.973,E2 7497.973} C_VEL
LIN {X 0,Y 154.381,Z 810.084,A -85,B 0,C 180,E1 7490.47,E2 7490.47} C_VEL
LIN {X 0,Y 153.664,Z 814.529,A -85,B 0,C 180,E1 7483.163,E2 7483.163} C_VEL
LIN {X 0,Y 154.477,Z 817.146,A -85,B 0,C 180,E1 7476.317,E2 7476.317} C_VEL
LIN {X 0,Y 155.33,Z 818.002,A -85,B 0,C 180,E1 7471.475,E2 7471.475} C_VEL
LIN {X 0,Y 155.288,Z 817.963,A -85,B 0,C 180,E1 7468.155,E2 7468.155} C_VEL
LIN {X 0,Y 154.41,Z 817.036,A -85,B 0,C 180,E1 7463.307,E2 7463.307} C_VEL
LIN {X 0,Y 153.66,Z 814.299,A -85,B 0,C 180,E1 7456.453,E2 7456.453} C_VEL
LIN {X 0,Y 154.477,Z 809.738,A -85,B 0,C 180,E1 7449.146,E2 7449.146} C_VEL
LIN {X 0,Y 157.4,Z 803.431,A -85,B 0,C 180,E1 7441.962,E2 7441.962} C_VEL
LIN {X 0,Y 162.907,Z 794.707,A -85,B 0,C 180,E1 7434.715,E2 7434.715} C_VEL
LIN {X 0,Y 170.226,Z 784.474,A -85,B 0,C 180,E1 7428.417,E2 7428.417} C_VEL
LIN {X 0,Y 179.072,Z 772.527,A -85,B 0,C 180,E1 7422.936,E2 7422.936} C_VEL
LIN {X 0,Y 188.874,Z 758.936,A -85,B 0,C 180,E1 7418.27,E2 7418.27} C_VEL
LIN {X 0,Y 198.905,Z 744.208,A -85,B 0,C 180,E1 7414.475,E2 7414.475} C_VEL
LIN {X 0,Y 208.956,Z 728.077,A -85,B 0,C 180,E1 7411.339,E2 7411.339} C_VEL
LIN {X 0,Y 218.658,Z 710.63,A -85,B 0,C 180,E1 7408.784,E2 7408.784} C_VEL
LIN {X 0,Y 227.411,Z 692.631,A -85,B 0,C 180,E1 7406.81,E2 7406.81} C_VEL
LIN {X 0,Y 235.429,Z 673.259,A -85,B 0,C 180,E1 7405.234,E2 7405.234} C_VEL
LIN {X 0,Y 242.213,Z 653.162,A -85,B 0,C 180,E1 7404.035,E2 7404.035} C_VEL
LIN {X 0,Y 247.571,Z 632.171,A -85,B 0,C 180,E1 7403.106,E2 7403.106} C_VEL
LIN {X 0,Y 251.245,Z 610.843,A -85,B 0,C 180,E1 7402.414,E2 7402.414} C_VEL
LIN {X 0,Y 263.553,Z 481.54,A -85,B 0,C 180,E1 7399.473,E2 7399.473} C_VEL
LIN {X 0,Y 259.34,Z 471.766,A -85,B 0,C 180,E1 7396.346,E2 7396.346} C_VEL
LIN {X 0,Y 255.173,Z 462.689,A -85,B 0,C 180,E1 7392.617,E2 7392.617} C_VEL
LIN {X 0,Y 251.911,Z 456.072,A -85,B 0,C 180,E1 7388.904,E2 7388.904} C_VEL
LIN {X 0,Y 249.48,Z 451.09,A -85,B 0,C 180,E1 7385.058,E2 7385.058} C_VEL
LIN {X 0,Y 247.82,Z 447.463,A -85,B 0,C 180,E1 7380.462,E2 7380.462} C_VEL
LIN {X 0,Y 247.462,Z 446.709,A -85,B 0,C 180,E1 7375.132,E2 7375.132} C_VEL
LIN {X 0,Y 248.791,Z 447.765,A -85,B 0,C 180,E1 7370.282,E2 7370.282} C_VEL
LIN {X 0,Y 251.559,Z 452.405,A -85,B 0,C 180,E1 7365.381,E2 7365.381} C_VEL
LIN {X 0,Y 254.284,Z 457.06,A -85,B 0,C 180,E1 7362.139,E2 7362.139} C_VEL
LIN {X 0,Y 257.727,Z 463.073,A -85,B 0,C 180,E1 7358.91,E2 7358.91} C_VEL
LIN {X 0,Y 261.996,Z 471.32,A -85,B 0,C 180,E1 7355.599,E2 7355.599} C_VEL
LIN {X 0,Y 263.551,Z 474.897,A -85,B 0,C 180,E1 7354.498,E2 7354.498} C_VEL
LIN {X 0,Y 254.321,Z 580.204,A -85,B 0,C 180,E1 7352.19,E2 7352.19} C_VEL
LIN {X 0,Y 251.971,Z 599.566,A -85,B 0,C 180,E1 7351.512,E2 7351.512} C_VEL
LIN {X 0,Y 248.294,Z 618.521,A -85,B 0,C 180,E1 7350.574,E2 7350.574} C_VEL
LIN {X 0,Y 243.3,Z 637.125,A -85,B 0,C 180,E1 7349.339,E2 7349.339} C_VEL
LIN {X 0,Y 237.016,Z 655.319,A -85,B 0,C 180,E1 7347.757,E2 7347.757} C_VEL
LIN {X 0,Y 229.638,Z 672.656,A -85,B 0,C 180,E1 7345.817,E2 7345.817} C_VEL
LIN {X 0,Y 221.442,Z 688.842,A -85,B 0,C 180,E1 7343.483,E2 7343.483} C_VEL
LIN {X 0,Y 212.56,Z 703.893,A -85,B 0,C 180,E1 7340.694,E2 7340.694} C_VEL
LIN {X 0,Y 203.521,Z 717.348,A -85,B 0,C 180,E1 7337.468,E2 7337.468} C_VEL
LIN {X 0,Y 194.218,Z 729.672,A -85,B 0,C 180,E1 7333.617,E2 7333.617} C_VEL
LIN {X 0,Y 185.224,Z 740.445,A -85,B 0,C 180,E1 7329.165,E2 7329.165} C_VEL
LIN {X 0,Y 176.868,Z 749.676,A -85,B 0,C 180,E1 7324.031,E2 7324.031} C_VEL
LIN {X 0,Y 169.47,Z 757.345,A -85,B 0,C 180,E1 7318.163,E2 7318.163} C_VEL
LIN {X 0,Y 163.427,Z 763.382,A -85,B 0,C 180,E1 7311.535,E2 7311.535} C_VEL
LIN {X 0,Y 159.252,Z 767.538,A -85,B 0,C 180,E1 7304.544,E2 7304.544} C_VEL
LIN {X 0,Y 156.86,Z 769.974,A -85,B 0,C 180,E1 7297.324,E2 7297.324} C_VEL
LIN {X 0,Y 156.11,Z 770.782,A -85,B 0,C 180,E1 7290,E2 7290} C_VEL
LIN {X 0,Y 156.844,Z 770.007,A -85,B 0,C 180,E1 7282.675,E2 7282.675} C_VEL
LIN {X 0,Y 159.218,Z 767.61,A -85,B 0,C 180,E1 7275.452,E2 7275.452} C_VEL
LIN {X 0,Y 163.375,Z 763.49,A -85,B 0,C 180,E1 7268.458,E2 7268.458} C_VEL
LIN {X 0,Y 169.4,Z 757.502,A -85,B 0,C 180,E1 7261.825,E2 7261.825} C_VEL
LIN {X 0,Y 176.785,Z 749.885,A -85,B 0,C 180,E1 7255.951,E2 7255.951} C_VEL
LIN {X 0,Y 185.13,Z 740.702,A -85,B 0,C 180,E1 7250.811,E2 7250.811} C_VEL
LIN {X 0,Y 194.118,Z 729.979,A -85,B 0,C 180,E1 7246.355,E2 7246.355} C_VEL
LIN {X 0,Y 203.414,Z 717.718,A -85,B 0,C 180,E1 7242.499,E2 7242.499} C_VEL
LIN {X 0,Y 212.774,Z 703.843,A -85,B 0,C 180,E1 7239.164,E2 7239.164} C_VEL
LIN {X 0,Y 221.669,Z 688.775,A -85,B 0,C 180,E1 7236.379,E2 7236.379} C_VEL
LIN {X 0,Y 229.879,Z 672.569,A -85,B 0,C 180,E1 7234.049,E2 7234.049} C_VEL
LIN {X 0,Y 237.266,Z 655.21,A -85,B 0,C 180,E1 7232.113,E2 7232.113} C_VEL
LIN {X 0,Y 243.69,Z 636.573,A -85,B 0,C 180,E1 7230.503,E2 7230.503} C_VEL
LIN {X 0,Y 248.705,Z 617.715,A -85,B 0,C 180,E1 7229.265,E2 7229.265} C_VEL
LIN {X 0,Y 252.48,Z 597.798,A -85,B 0,C 180,E1 7228.299,E2 7228.299} C_VEL
LIN {X 0,Y 254.79,Z 577.427,A -85,B 0,C 180,E1 7227.618,E2 7227.618} C_VEL
LIN {X 0,Y 263.739,Z 474.717,A -85,B 0,C 180,E1 7225.366,E2 7225.366} C_VEL
LIN {X 0,Y 259.552,Z 466.229,A -85,B 0,C 180,E1 7222.3,E2 7222.3} C_VEL
LIN {X 0,Y 255.458,Z 458.844,A -85,B 0,C 180,E1 7218.71,E2 7218.71} C_VEL
LIN {X 0,Y 252.926,Z 454.585,A -85,B 0,C 180,E1 7215.947,E2 7215.947} C_VEL
LIN {X 0,Y 251.182,Z 451.572,A -85,B 0,C 180,E1 7213.584,E2 7213.584} C_VEL
LIN {X 0,Y 248.738,Z 447.601,A -85,B 0,C 180,E1 7208.787,E2 7208.787} C_VEL
LIN {X 0,Y 247.663,Z 446.989,A -85,B 0,C 180,E1 7203.009,E2 7203.009} C_VEL
LIN {X 0,Y 248.204,Z 447.955,A -85,B 0,C 180,E1 7199.077,E2 7199.077} C_VEL
LIN {X 0,Y 250.085,Z 452.118,A -85,B 0,C 180,E1 7194.264,E2 7194.264} C_VEL
LIN {X 0,Y 252.656,Z 457.359,A -85,B 0,C 180,E1 7190.433,E2 7190.433} C_VEL
LIN {X 0,Y 256.105,Z 464.467,A -85,B 0,C 180,E1 7186.683,E2 7186.683} C_VEL
LIN {X 0,Y 260.086,Z 473.128,A -85,B 0,C 180,E1 7183.243,E2 7183.243} C_VEL
LIN {X 0,Y 263.781,Z 481.757,A -85,B 0,C 180,E1 7180.523,E2 7180.523} C_VEL
LIN {X 0,Y 257.975,Z 543.047,A -85,B 0,C 180,E1 7179.173,E2 7179.173} C_VEL
LIN {X 0,Y 256.837,Z 550.728,A -85,B 0,C 180,E1 7179.207,E2 7179.207} C_VEL
LIN {X 0,Y 252.404,Z 571.174,A -85,B 0,C 180,E1 7180.036,E2 7180.036} C_VEL
LIN {X 0,Y 251.472,Z 577.768,A -85,B 0,C 180,E1 7180.05,E2 7180.05} C_VEL
LIN {X 0,Y 247.799,Z 612.659,A -85,B 0,C 180,E1 7179.224,E2 7179.224} C_VEL
LIN {X 0,Y 244.011,Z 633.123,A -85,B 0,C 180,E1 7178.555,E2 7178.555} C_VEL
LIN {X 0,Y 238.821,Z 652.717,A -85,B 0,C 180,E1 7177.702,E2 7177.702} C_VEL
LIN {X 0,Y 232.091,Z 672.178,A -85,B 0,C 180,E1 7176.576,E2 7176.576} C_VEL
LIN {X 0,Y 223.86,Z 691.55,A -85,B 0,C 180,E1 7175.048,E2 7175.048} C_VEL
LIN {X 0,Y 214.706,Z 709.79,A -85,B 0,C 180,E1 7173.096,E2 7173.096} C_VEL
LIN {X 0,Y 204.803,Z 726.974,A -85,B 0,C 180,E1 7170.624,E2 7170.624} C_VEL
LIN {X 0,Y 194.35,Z 743.09,A -85,B 0,C 180,E1 7167.532,E2 7167.532} C_VEL
LIN {X 0,Y 183.658,Z 758.072,A -85,B 0,C 180,E1 7163.679,E2 7163.679} C_VEL
LIN {X 0,Y 173.438,Z 771.461,A -85,B 0,C 180,E1 7159.041,E2 7159.041} C_VEL
LIN {X 0,Y 164.084,Z 783.3,A -85,B 0,C 180,E1 7153.516,E2 7153.516} C_VEL
LIN {X 0,Y 156.127,Z 793.575,A -85,B 0,C 180,E1 7147.011,E2 7147.011} C_VEL
LIN {X 0,Y 150.1,Z 802.221,A -85,B 0,C 180,E1 7139.533,E2 7139.533} C_VEL
LIN {X 0,Y 146.653,Z 808.825,A -85,B 0,C 180,E1 7131.602,E2 7131.602} C_VEL
LIN {X 0,Y 145.702,Z 813.285,A -85,B 0,C 180,E1 7123.897,E2 7123.897} C_VEL
LIN {X 0,Y 146.466,Z 815.921,A -85,B 0,C 180,E1 7116.664,E2 7116.664} C_VEL
LIN {X 0,Y 147.401,Z 816.797,A -85,B 0,C 180,E1 7111.555,E2 7111.555} C_VEL
LIN {X 0,Y 147.351,Z 816.757,A -85,B 0,C 180,E1 7108.056,E2 7108.056} C_VEL
LIN {X 0,Y 146.324,Z 815.709,A -85,B 0,C 180,E1 7102.54,E2 7102.54} C_VEL
LIN {X 0,Y 145.711,Z 812.851,A -85,B 0,C 180,E1 7095.292,E2 7095.292} C_VEL
LIN {X 0,Y 147.013,Z 807.873,A -85,B 0,C 180,E1 7087.191,E2 7087.191} C_VEL
LIN {X 0,Y 150.608,Z 801.312,A -85,B 0,C 180,E1 7079.659,E2 7079.659} C_VEL
LIN {X 0,Y 156.491,Z 792.975,A -85,B 0,C 180,E1 7072.63,E2 7072.63} C_VEL
LIN {X 0,Y 164.082,Z 783.179,A -85,B 0,C 180,E1 7066.48,E2 7066.48} C_VEL
LIN {X 0,Y 173.432,Z 771.32,A -85,B 0,C 180,E1 7060.956,E2 7060.956} C_VEL
LIN {X 0,Y 183.65,Z 757.9,A -85,B 0,C 180,E1 7056.318,E2 7056.318} C_VEL
LIN {X 0,Y 194.34,Z 742.872,A -85,B 0,C 180,E1 7052.463,E2 7052.463} C_VEL
LIN {X 0,Y 204.792,Z 726.711,A -85,B 0,C 180,E1 7049.37,E2 7049.37} C_VEL
LIN {X 0,Y 214.696,Z 709.474,A -85,B 0,C 180,E1 7046.899,E2 7046.899} C_VEL
LIN {X 0,Y 223.85,Z 691.159,A -85,B 0,C 180,E1 7044.946,E2 7044.946} C_VEL
LIN {X 0,Y 231.87,Z 672.23,A -85,B 0,C 180,E1 7043.455,E2 7043.455} C_VEL
LIN {X 0,Y 238.81,Z 652.104,A -85,B 0,C 180,E1 7042.292,E2 7042.292} C_VEL
LIN {X 0,Y 244.27,Z 631.118,A -85,B 0,C 180,E1 7041.391,E2 7041.391} C_VEL
LIN {X 0,Y 248,Z 609.891,A -85,B 0,C 180,E1 7040.719,E2 7040.719} C_VEL
LIN {X 0,Y 260.144,Z 485.777,A -85,B 0,C 180,E1 7037.938,E2 7037.938} C_VEL
LIN {X 0,Y 256.385,Z 476.76,A -85,B 0,C 180,E1 7034.857,E2 7034.857} C_VEL
LIN {X 0,Y 252.994,Z 469.085,A -85,B 0,C 180,E1 7031.512,E2 7031.512} C_VEL
LIN {X 0,Y 250.154,Z 462.889,A -85,B 0,C 180,E1 7027.926,E2 7027.926} C_VEL
LIN {X 0,Y 248.129,Z 458.615,A -85,B 0,C 180,E1 7024.391,E2 7024.391} C_VEL
LIN {X 0,Y 246.784,Z 455.352,A -85,B 0,C 180,E1 7020.232,E2 7020.232} C_VEL
LIN {X 0,Y 246.49,Z 454.651,A -85,B 0,C 180,E1 7015.113,E2 7015.113} C_VEL
LIN {X 0,Y 247.721,Z 455.697,A -85,B 0,C 180,E1 7010.474,E2 7010.474} C_VEL
LIN {X 0,Y 250.266,Z 460.124,A -85,B 0,C 180,E1 7005.776,E2 7005.776} C_VEL
LIN {X 0,Y 252.789,Z 464.632,A -85,B 0,C 180,E1 7002.624,E2 7002.624} C_VEL
LIN {X 0,Y 256.044,Z 470.619,A -85,B 0,C 180,E1 6999.423,E2 6999.423} C_VEL
LIN {X 0,Y 259.951,Z 478.537,A -85,B 0,C 180,E1 6996.244,E2 6996.244} C_VEL
LIN {X 0,Y 260.188,Z 479.476,A -85,B 0,C 180,E1 6996.034,E2 6996.034} C_VEL
LIN {X 0,Y 251.001,Z 580.966,A -85,B 0,C 180,E1 6993.832,E2 6993.832} C_VEL
LIN {X 0,Y 248.557,Z 600.417,A -85,B 0,C 180,E1 6993.157,E2 6993.157} C_VEL
LIN {X 0,Y 244.717,Z 619.559,A -85,B 0,C 180,E1 6992.221,E2 6992.221} C_VEL
LIN {X 0,Y 239.517,Z 638.294,A -85,B 0,C 180,E1 6990.989,E2 6990.989} C_VEL
LIN {X 0,Y 233.278,Z 655.875,A -85,B 0,C 180,E1 6989.484,E2 6989.484} C_VEL
LIN {X 0,Y 225.771,Z 673.077,A -85,B 0,C 180,E1 6987.597,E2 6987.597} C_VEL
LIN {X 0,Y 217.188,Z 689.557,A -85,B 0,C 180,E1 6985.258,E2 6985.258} C_VEL
LIN {X 0,Y 207.98,Z 704.672,A -85,B 0,C 180,E1 6982.487,E2 6982.487} C_VEL
LIN {X 0,Y 198.259,Z 718.598,A -85,B 0,C 180,E1 6979.153,E2 6979.153} C_VEL
LIN {X 0,Y 188.564,Z 730.905,A -85,B 0,C 180,E1 6975.277,E2 6975.277} C_VEL
LIN {X 0,Y 179.149,Z 741.668,A -85,B 0,C 180,E1 6970.766,E2 6970.766} C_VEL
LIN {X 0,Y 170.352,Z 750.892,A -85,B 0,C 180,E1 6965.525,E2 6965.525} C_VEL
LIN {X 0,Y 162.518,Z 758.555,A -85,B 0,C 180,E1 6959.483,E2 6959.483} C_VEL
LIN {X 0,Y 156.075,Z 764.587,A -85,B 0,C 180,E1 6952.604,E2 6952.604} C_VEL
LIN {X 0,Y 151.594,Z 768.742,A -85,B 0,C 180,E1 6945.297,E2 6945.297} C_VEL
LIN {X 0,Y 149.013,Z 771.177,A -85,B 0,C 180,E1 6937.712,E2 6937.712} C_VEL
LIN {X 0,Y 148.201,Z 771.984,A -85,B 0,C 180,E1 6930,E2 6930} C_VEL
LIN {X 0,Y 148.996,Z 771.208,A -85,B 0,C 180,E1 6922.287,E2 6922.287} C_VEL
LIN {X 0,Y 151.559,Z 768.813,A -85,B 0,C 180,E1 6914.7,E2 6914.7} C_VEL
LIN {X 0,Y 156.133,Z 764.602,A -85,B 0,C 180,E1 6907.246,E2 6907.246} C_VEL
LIN {X 0,Y 162.449,Z 758.708,A -85,B 0,C 180,E1 6900.503,E2 6900.503} C_VEL
LIN {X 0,Y 170.27,Z 751.095,A -85,B 0,C 180,E1 6894.456,E2 6894.456} C_VEL
LIN {X 0,Y 179.056,Z 741.918,A -85,B 0,C 180,E1 6889.208,E2 6889.208} C_VEL
LIN {X 0,Y 188.466,Z 731.205,A -85,B 0,C 180,E1 6884.693,E2 6884.693} C_VEL
LIN {X 0,Y 198.154,Z 718.96,A -85,B 0,C 180,E1 6880.812,E2 6880.812} C_VEL
LIN {X 0,Y 207.872,Z 705.108,A -85,B 0,C 180,E1 6877.475,E2 6877.475} C_VEL
LIN {X 0,Y 217.158,Z 689.944,A -85,B 0,C 180,E1 6874.679,E2 6874.679} C_VEL
LIN {X 0,Y 225.558,Z 673.92,A -85,B 0,C 180,E1 6872.39,E2 6872.39} C_VEL
LIN {X 0,Y 233.175,Z 656.639,A -85,B 0,C 180,E1 6870.473,E2 6870.473} C_VEL
LIN {X 0,Y 239.573,Z 638.784,A -85,B 0,C 180,E1 6868.934,E2 6868.934} C_VEL
LIN {X 0,Y 244.673,Z 620.585,A -85,B 0,C 180,E1 6867.727,E2 6867.727} C_VEL
LIN {X 0,Y 248.553,Z 601.667,A -85,B 0,C 180,E1 6866.784,E2 6866.784} C_VEL
LIN {X 0,Y 251.088,Z 582.292,A -85,B 0,C 180,E1 6866.096,E2 6866.096} C_VEL
LIN {X 0,Y 257.593,Z 510.007,A -85,B 0,C 180,E1 6864.486,E2 6864.486} C_VEL
LIN {X 0,Y 260.403,Z 479.233,A -85,B 0,C 180,E1 6863.831,E2 6863.831} C_VEL
LIN {X 0,Y 256.523,Z 471.34,A -85,B 0,C 180,E1 6860.702,E2 6860.702} C_VEL
LIN {X 0,Y 253.207,Z 465.166,A -85,B 0,C 180,E1 6857.465,E2 6857.465} C_VEL
LIN {X 0,Y 251.234,Z 461.709,A -85,B 0,C 180,E1 6855.111,E2 6855.111} C_VEL
LIN {X 0,Y 249.755,Z 459.117,A -85,B 0,C 180,E1 6852.956,E2 6852.956} C_VEL
LIN {X 0,Y 247.684,Z 455.499,A -85,B 0,C 180,E1 6848.591,E2 6848.591} C_VEL
LIN {X 0,Y 246.69,Z 454.93,A -85,B 0,C 180,E1 6843.021,E2 6843.021} C_VEL
LIN {X 0,Y 247.153,Z 455.842,A -85,B 0,C 180,E1 6839.305,E2 6839.305} C_VEL
LIN {X 0,Y 248.83,Z 459.798,A -85,B 0,C 180,E1 6834.698,E2 6834.698} C_VEL
LIN {X 0,Y 251.269,Z 465.053,A -85,B 0,C 180,E1 6830.842,E2 6830.842} C_VEL
LIN {X 0,Y 254.479,Z 472.046,A -85,B 0,C 180,E1 6827.174,E2 6827.174} C_VEL
LIN {X 0,Y 258.364,Z 481.072,A -85,B 0,C 180,E1 6823.648,E2 6823.648} C_VEL
LIN {X 0,Y 260.366,Z 486.215,A -85,B 0,C 180,E1 6822.046,E2 6822.046} C_VEL
LIN {X 0,Y 251.472,Z 577.768,A -85,B 0,C 180,E1 6820.05,E2 6820.05} C_VEL
LIN {X 0,Y 250.372,Z 585.459,A -85,B 0,C 180,E1 6820.096,E2 6820.096} C_VEL
LIN {X 0,Y 245.891,Z 605.89,A -85,B 0,C 180,E1 6820.959,E2 6820.959} C_VEL
LIN {X 0,Y 244.663,Z 612.43,A -85,B 0,C 180,E1 6820.942,E2 6820.942} C_VEL
LIN {X 0,Y 240.783,Z 632.702,A -85,B 0,C 180,E1 6820.293,E2 6820.293} C_VEL
LIN {X 0,Y 235.429,Z 652.333,A -85,B 0,C 180,E1 6819.46,E2 6819.46} C_VEL
LIN {X 0,Y 228.669,Z 671.403,A -85,B 0,C 180,E1 6818.391,E2 6818.391} C_VEL
LIN {X 0,Y 220.544,Z 690.09,A -85,B 0,C 180,E1 6816.969,E2 6816.969} C_VEL
LIN {X 0,Y 211.054,Z 708.526,A -85,B 0,C 180,E1 6815.063,E2 6815.063} C_VEL
LIN {X 0,Y 200.748,Z 725.851,A -85,B 0,C 180,E1 6812.634,E2 6812.634} C_VEL
LIN {X 0,Y 189.676,Z 742.276,A -85,B 0,C 180,E1 6809.525,E2 6809.525} C_VEL
LIN {X 0,Y 178.87,Z 756.768,A -85,B 0,C 180,E1 6805.82,E2 6805.82} C_VEL
LIN {X 0,Y 168.095,Z 770.168,A -85,B 0,C 180,E1 6801.186,E2 6801.186} C_VEL
LIN {X 0,Y 158.139,Z 782.016,A -85,B 0,C 180,E1 6795.597,E2 6795.597} C_VEL
LIN {X 0,Y 149.543,Z 792.296,A -85,B 0,C 180,E1 6788.938,E2 6788.938} C_VEL
LIN {X 0,Y 142.909,Z 800.951,A -85,B 0,C 180,E1 6781.179,E2 6781.179} C_VEL
LIN {X 0,Y 138.985,Z 807.564,A -85,B 0,C 180,E1 6772.859,E2 6772.859} C_VEL
LIN {X 0,Y 137.753,Z 812.039,A -85,B 0,C 180,E1 6764.716,E2 6764.716} C_VEL
LIN {X 0,Y 138.445,Z 814.695,A -85,B 0,C 180,E1 6757.052,E2 6757.052} C_VEL
LIN {X 0,Y 139.466,Z 815.591,A -85,B 0,C 180,E1 6751.643,E2 6751.643} C_VEL
LIN {X 0,Y 139.466,Z 815.586,A -85,B 0,C 180,E1 6748.357,E2 6748.357} C_VEL
LIN {X 0,Y 138.448,Z 814.681,A -85,B 0,C 180,E1 6742.948,E2 6742.948} C_VEL
LIN {X 0,Y 137.765,Z 811.803,A -85,B 0,C 180,E1 6734.853,E2 6734.853} C_VEL
LIN {X 0,Y 139.121,Z 807.214,A -85,B 0,C 180,E1 6726.717,E2 6726.717} C_VEL
LIN {X 0,Y 142.907,Z 800.885,A -85,B 0,C 180,E1 6718.82,E2 6718.82} C_VEL
LIN {X 0,Y 149.54,Z 792.205,A -85,B 0,C 180,E1 6711.061,E2 6711.061} C_VEL
LIN {X 0,Y 158.135,Z 781.896,A -85,B 0,C 180,E1 6704.401,E2 6704.401} C_VEL
LIN {X 0,Y 168.089,Z 770.02,A -85,B 0,C 180,E1 6698.811,E2 6698.811} C_VEL
LIN {X 0,Y 178.861,Z 756.587,A -85,B 0,C 180,E1 6694.176,E2 6694.176} C_VEL
LIN {X 0,Y 190.029,Z 741.535,A -85,B 0,C 180,E1 6690.358,E2 6690.358} C_VEL
LIN {X 0,Y 200.882,Z 725.341,A -85,B 0,C 180,E1 6687.323,E2 6687.323} C_VEL
LIN {X 0,Y 210.959,Z 708.352,A -85,B 0,C 180,E1 6684.949,E2 6684.949} C_VEL
LIN {X 0,Y 220.118,Z 690.564,A -85,B 0,C 180,E1 6683.102,E2 6683.102} C_VEL
LIN {X 0,Y 228.119,Z 672.224,A -85,B 0,C 180,E1 6681.692,E2 6681.692} C_VEL
LIN {X 0,Y 234.988,Z 653.026,A -85,B 0,C 180,E1 6680.6,E2 6680.6} C_VEL
LIN {X 0,Y 240.448,Z 633.199,A -85,B 0,C 180,E1 6679.749,E2 6679.749} C_VEL
LIN {X 0,Y 244.372,Z 612.887,A -85,B 0,C 180,E1 6679.092,E2 6679.092} C_VEL
LIN {X 0,Y 247.847,Z 581.803,A -85,B 0,C 180,E1 6678.357,E2 6678.357} C_VEL
LIN {X 0,Y 256.947,Z 490.156,A -85,B 0,C 180,E1 6676.386,E2 6676.386} C_VEL
LIN {X 0,Y 253.38,Z 481.296,A -85,B 0,C 180,E1 6673.114,E2 6673.114} C_VEL
LIN {X 0,Y 250.863,Z 475.413,A -85,B 0,C 180,E1 6670.332,E2 6670.332} C_VEL
LIN {X 0,Y 248.668,Z 470.294,A -85,B 0,C 180,E1 6667.276,E2 6667.276} C_VEL
LIN {X 0,Y 246.914,Z 466.316,A -85,B 0,C 180,E1 6663.947,E2 6663.947} C_VEL
LIN {X 0,Y 245.743,Z 463.239,A -85,B 0,C 180,E1 6660,E2 6660} C_VEL
LIN {X 0,Y 245.547,Z 462.608,A -85,B 0,C 180,E1 6654.86,E2 6654.86} C_VEL
LIN {X 0,Y 246.654,Z 463.625,A -85,B 0,C 180,E1 6650.668,E2 6650.668} C_VEL
LIN {X 0,Y 248.984,Z 467.843,A -85,B 0,C 180,E1 6646.176,E2 6646.176} C_VEL
LIN {X 0,Y 251.404,Z 472.39,A -85,B 0,C 180,E1 6643.003,E2 6643.003} C_VEL
LIN {X 0,Y 254.563,Z 478.529,A -85,B 0,C 180,E1 6639.779,E2 6639.779} C_VEL
LIN {X 0,Y 257.045,Z 483.834,A -85,B 0,C 180,E1 6637.615,E2 6637.615} C_VEL
LIN {X 0,Y 247.915,Z 581.507,A -85,B 0,C 180,E1 6635.523,E2 6635.523} C_VEL
LIN {X 0,Y 245.389,Z 601.071,A -85,B 0,C 180,E1 6634.855,E2 6634.855} C_VEL
LIN {X 0,Y 241.502,Z 620.015,A -85,B 0,C 180,E1 6633.947,E2 6633.947} C_VEL
LIN {X 0,Y 236.186,Z 638.749,A -85,B 0,C 180,E1 6632.745,E2 6632.745} C_VEL
LIN {X 0,Y 229.38,Z 657.321,A -85,B 0,C 180,E1 6631.179,E2 6631.179} C_VEL
LIN {X 0,Y 221.535,Z 674.663,A -85,B 0,C 180,E1 6629.29,E2 6629.29} C_VEL
LIN {X 0,Y 212.789,Z 690.868,A -85,B 0,C 180,E1 6627.005,E2 6627.005} C_VEL
LIN {X 0,Y 203.265,Z 705.946,A -85,B 0,C 180,E1 6624.254,E2 6624.254} C_VEL
LIN {X 0,Y 193.177,Z 719.844,A -85,B 0,C 180,E1 6620.928,E2 6620.928} C_VEL
LIN {X 0,Y 183.078,Z 732.135,A -85,B 0,C 180,E1 6617.038,E2 6617.038} C_VEL
LIN {X 0,Y 173.224,Z 742.889,A -85,B 0,C 180,E1 6612.478,E2 6612.478} C_VEL
LIN {X 0,Y 163.96,Z 752.107,A -85,B 0,C 180,E1 6607.136,E2 6607.136} C_VEL
LIN {X 0,Y 155.661,Z 759.765,A -85,B 0,C 180,E1 6600.921,E2 6600.921} C_VEL
LIN {X 0,Y 148.783,Z 765.793,A -85,B 0,C 180,E1 6593.779,E2 6593.779} C_VEL
LIN {X 0,Y 143.964,Z 769.946,A -85,B 0,C 180,E1 6586.129,E2 6586.129} C_VEL
LIN {X 0,Y 141.173,Z 772.379,A -85,B 0,C 180,E1 6578.143,E2 6578.143} C_VEL
LIN {X 0,Y 140.292,Z 773.185,A -85,B 0,C 180,E1 6570,E2 6570} C_VEL
LIN {X 0,Y 141.156,Z 772.41,A -85,B 0,C 180,E1 6561.856,E2 6561.856} C_VEL
LIN {X 0,Y 143.929,Z 770.016,A -85,B 0,C 180,E1 6553.867,E2 6553.867} C_VEL
LIN {X 0,Y 148.729,Z 765.899,A -85,B 0,C 180,E1 6546.212,E2 6546.212} C_VEL
LIN {X 0,Y 155.591,Z 759.914,A -85,B 0,C 180,E1 6539.064,E2 6539.064} C_VEL
LIN {X 0,Y 163.879,Z 752.305,A -85,B 0,C 180,E1 6532.843,E2 6532.843} C_VEL
LIN {X 0,Y 173.131,Z 743.134,A -85,B 0,C 180,E1 6527.494,E2 6527.494} C_VEL
LIN {X 0,Y 182.982,Z 732.43,A -85,B 0,C 180,E1 6522.93,E2 6522.93} C_VEL
LIN {X 0,Y 193.075,Z 720.2,A -85,B 0,C 180,E1 6519.035,E2 6519.035} C_VEL
LIN {X 0,Y 203.161,Z 706.372,A -85,B 0,C 180,E1 6515.706,E2 6515.706} C_VEL
LIN {X 0,Y 212.685,Z 691.374,A -85,B 0,C 180,E1 6512.952,E2 6512.952} C_VEL
LIN {X 0,Y 221.287,Z 675.555,A -85,B 0,C 180,E1 6510.703,E2 6510.703} C_VEL
LIN {X 0,Y 228.902,Z 658.944,A -85,B 0,C 180,E1 6508.864,E2 6508.864} C_VEL
LIN {X 0,Y 235.329,Z 641.891,A -85,B 0,C 180,E1 6507.381,E2 6507.381} C_VEL
LIN {X 0,Y 240.875,Z 623.254,A -85,B 0,C 180,E1 6506.128,E2 6506.128} C_VEL
LIN {X 0,Y 245.108,Z 603.844,A -85,B 0,C 180,E1 6505.152,E2 6505.152} C_VEL
LIN {X 0,Y 247.888,Z 583.957,A -85,B 0,C 180,E1 6504.438,E2 6504.438} C_VEL
LIN {X 0,Y 253.734,Z 521.064,A -85,B 0,C 180,E1 6503.035,E2 6503.035} C_VEL
LIN {X 0,Y 257.195,Z 483.763,A -85,B 0,C 180,E1 6502.224,E2 6502.224} C_VEL
LIN {X 0,Y 253.712,Z 476.578,A -85,B 0,C 180,E1 6499.093,E2 6499.093} C_VEL
LIN {X 0,Y 250.608,Z 470.559,A -85,B 0,C 180,E1 6495.624,E2 6495.624} C_VEL
LIN {X 0,Y 248.499,Z 466.835,A -85,B 0,C 180,E1 6492.549,E2 6492.549} C_VEL
LIN {X 0,Y 246.632,Z 463.397,A -85,B 0,C 180,E1 6488.393,E2 6488.393} C_VEL
LIN {X 0,Y 245.708,Z 462.87,A -85,B 0,C 180,E1 6483.033,E2 6483.033} C_VEL
LIN {X 0,Y 246.106,Z 463.728,A -85,B 0,C 180,E1 6479.535,E2 6479.535} C_VEL
LIN {X 0,Y 247.641,Z 467.633,A -85,B 0,C 180,E1 6475.021,E2 6475.021} C_VEL
LIN {X 0,Y 249.902,Z 472.748,A -85,B 0,C 180,E1 6471.255,E2 6471.255} C_VEL
LIN {X 0,Y 252.815,Z 479.538,A -85,B 0,C 180,E1 6467.727,E2 6467.727} C_VEL
LIN {X 0,Y 256.4,Z 488.415,A -85,B 0,C 180,E1 6464.275,E2 6464.275} C_VEL
LIN {X 0,Y 257.139,Z 490.654,A -85,B 0,C 180,E1 6463.613,E2 6463.613} C_VEL
LIN {X 0,Y 245.047,Z 610.055,A -85,B 0,C 180,E1 6461.01,E2 6461.01} C_VEL
LIN {X 0,Y 244.663,Z 612.43,A -85,B 0,C 180,E1 6460.942,E2 6460.942} C_VEL
LIN {X 0,Y 243.019,Z 620.008,A -85,B 0,C 180,E1 6460.963,E2 6460.963} C_VEL
LIN {X 0,Y 236.846,Z 637.811,A -85,B 0,C 180,E1 6461.606,E2 6461.606} C_VEL
LIN {X 0,Y 234.337,Z 645.192,A -85,B 0,C 180,E1 6461.564,E2 6461.564} C_VEL
LIN {X 0,Y 234.022,Z 646.228,A -85,B 0,C 180,E1 6461.524,E2 6461.524} C_VEL
LIN {X 0,Y 227.43,Z 665.555,A -85,B 0,C 180,E1 6460.559,E2 6460.559} C_VEL
LIN {X 0,Y 219.189,Z 684.926,A -85,B 0,C 180,E1 6459.245,E2 6459.245} C_VEL
LIN {X 0,Y 209.883,Z 703.202,A -85,B 0,C 180,E1 6457.543,E2 6457.543} C_VEL
LIN {X 0,Y 199.515,Z 720.678,A -85,B 0,C 180,E1 6455.33,E2 6455.33} C_VEL
LIN {X 0,Y 188.277,Z 737.25,A -85,B 0,C 180,E1 6452.478,E2 6452.478} C_VEL
LIN {X 0,Y 177.173,Z 751.883,A -85,B 0,C 180,E1 6449.067,E2 6449.067} C_VEL
LIN {X 0,Y 166.211,Z 765.114,A -85,B 0,C 180,E1 6444.895,E2 6444.895} C_VEL
LIN {X 0,Y 155.772,Z 776.983,A -85,B 0,C 180,E1 6439.801,E2 6439.801} C_VEL
LIN {X 0,Y 146.309,Z 787.449,A -85,B 0,C 180,E1 6433.646,E2 6433.646} C_VEL
LIN {X 0,Y 138.442,Z 796.451,A -85,B 0,C 180,E1 6426.314,E2 6426.314} C_VEL
LIN {X 0,Y 133.041,Z 803.577,A -85,B 0,C 180,E1 6418.259,E2 6418.259} C_VEL
LIN {X 0,Y 130.135,Z 809.242,A -85,B 0,C 180,E1 6409.087,E2 6409.087} C_VEL
LIN {X 0,Y 129.976,Z 812.621,A -85,B 0,C 180,E1 6400.639,E2 6400.639} C_VEL
LIN {X 0,Y 131.211,Z 814.223,A -85,B 0,C 180,E1 6393.402,E2 6393.402} C_VEL
LIN {X 0,Y 131.671,Z 814.48,A -85,B 0,C 180,E1 6389.565,E2 6389.565} C_VEL
LIN {X 0,Y 130.744,Z 813.85,A -85,B 0,C 180,E1 6384.294,E2 6384.294} C_VEL
LIN {X 0,Y 129.807,Z 811.681,A -85,B 0,C 180,E1 6376.64,E2 6376.64} C_VEL
LIN {X 0,Y 130.727,Z 807.581,A -85,B 0,C 180,E1 6367.99,E2 6367.99} C_VEL
LIN {X 0,Y 134.463,Z 801.416,A -85,B 0,C 180,E1 6359.132,E2 6359.132} C_VEL
LIN {X 0,Y 140.678,Z 793.709,A -85,B 0,C 180,E1 6351.286,E2 6351.286} C_VEL
LIN {X 0,Y 149.409,Z 783.877,A -85,B 0,C 180,E1 6344.104,E2 6344.104} C_VEL
LIN {X 0,Y 159.903,Z 772.197,A -85,B 0,C 180,E1 6338.016,E2 6338.016} C_VEL
LIN {X 0,Y 170.874,Z 759.42,A -85,B 0,C 180,E1 6333.203,E2 6333.203} C_VEL
LIN {X 0,Y 182.255,Z 745.141,A -85,B 0,C 180,E1 6329.278,E2 6329.278} C_VEL
LIN {X 0,Y 193.273,Z 729.866,A -85,B 0,C 180,E1 6326.181,E2 6326.181} C_VEL
LIN {X 0,Y 203.564,Z 713.828,A -85,B 0,C 180,E1 6323.751,E2 6323.751} C_VEL
LIN {X 0,Y 213.225,Z 696.613,A -85,B 0,C 180,E1 6321.807,E2 6321.807} C_VEL
LIN {X 0,Y 221.836,Z 678.694,A -85,B 0,C 180,E1 6320.307,E2 6320.307} C_VEL
LIN {X 0,Y 229.62,Z 659.128,A -85,B 0,C 180,E1 6319.112,E2 6319.112} C_VEL
LIN {X 0,Y 235.854,Z 639.101,A -85,B 0,C 180,E1 6318.2,E2 6318.2} C_VEL
LIN {X 0,Y 240.515,Z 618.355,A -85,B 0,C 180,E1 6317.488,E2 6317.488} C_VEL
LIN {X 0,Y 243.51,Z 596.855,A -85,B 0,C 180,E1 6316.942,E2 6316.942} C_VEL
LIN {X 0,Y 253.906,Z 494.611,A -85,B 0,C 180,E1 6314.772,E2 6314.772} C_VEL
LIN {X 0,Y 250.65,Z 486.073,A -85,B 0,C 180,E1 6311.388,E2 6311.388} C_VEL
LIN {X 0,Y 247.772,Z 479.008,A -85,B 0,C 180,E1 6307.536,E2 6307.536} C_VEL
LIN {X 0,Y 245.813,Z 474.192,A -85,B 0,C 180,E1 6303.731,E2 6303.731} C_VEL
LIN {X 0,Y 244.707,Z 471.127,A -85,B 0,C 180,E1 6299.765,E2 6299.765} C_VEL
LIN {X 0,Y 244.572,Z 470.551,A -85,B 0,C 180,E1 6294.839,E2 6294.839} C_VEL
LIN {X 0,Y 245.601,Z 471.552,A -85,B 0,C 180,E1 6290.864,E2 6290.864} C_VEL
LIN {X 0,Y 247.777,Z 475.718,A -85,B 0,C 180,E1 6286.464,E2 6286.464} C_VEL
LIN {X 0,Y 249.935,Z 479.958,A -85,B 0,C 180,E1 6283.498,E2 6283.498} C_VEL
LIN {X 0,Y 253.156,Z 486.57,A -85,B 0,C 180,E1 6280.07,E2 6280.07} C_VEL
LIN {X 0,Y 254.035,Z 488.817,A -85,B 0,C 180,E1 6279.22,E2 6279.22} C_VEL
LIN {X 0,Y 245.027,Z 582.268,A -85,B 0,C 180,E1 6277.248,E2 6277.248} C_VEL
LIN {X 0,Y 242.417,Z 601.854,A -85,B 0,C 180,E1 6276.59,E2 6276.59} C_VEL
LIN {X 0,Y 238.437,Z 620.741,A -85,B 0,C 180,E1 6275.704,E2 6275.704} C_VEL
LIN {X 0,Y 233.082,Z 639.179,A -85,B 0,C 180,E1 6274.55,E2 6274.55} C_VEL
LIN {X 0,Y 226.079,Z 657.877,A -85,B 0,C 180,E1 6273.016,E2 6273.016} C_VEL
LIN {X 0,Y 217.997,Z 675.305,A -85,B 0,C 180,E1 6271.165,E2 6271.165} C_VEL
LIN {X 0,Y 208.969,Z 691.58,A -85,B 0,C 180,E1 6268.919,E2 6268.919} C_VEL
LIN {X 0,Y 199.111,Z 706.721,A -85,B 0,C 180,E1 6266.207,E2 6266.207} C_VEL
LIN {X 0,Y 188.972,Z 720.256,A -85,B 0,C 180,E1 6263.027,E2 6263.027} C_VEL
LIN {X 0,Y 178.413,Z 732.669,A -85,B 0,C 180,E1 6259.16,E2 6259.16} C_VEL
LIN {X 0,Y 168.042,Z 743.531,A -85,B 0,C 180,E1 6254.595,E2 6254.595} C_VEL
LIN {X 0,Y 158.215,Z 752.852,A -85,B 0,C 180,E1 6249.194,E2 6249.194} C_VEL
LIN {X 0,Y 149.331,Z 760.614,A -85,B 0,C 180,E1 6242.842,E2 6242.842} C_VEL
LIN {X 0,Y 141.877,Z 766.753,A -85,B 0,C 180,E1 6235.46,E2 6235.46} C_VEL
LIN {X 0,Y 136.579,Z 770.991,A -85,B 0,C 180,E1 6227.466,E2 6227.466} C_VEL
LIN {X 0,Y 133.342,Z 773.581,A -85,B 0,C 180,E1 6218.625,E2 6218.625} C_VEL
LIN {X 0,Y 132.383,Z 774.387,A -85,B 0,C 180,E1 6210,E2 6210} C_VEL
LIN {X 0,Y 133.325,Z 773.612,A -85,B 0,C 180,E1 6201.374,E2 6201.374} C_VEL
LIN {X 0,Y 136.332,Z 771.219,A -85,B 0,C 180,E1 6192.941,E2 6192.941} C_VEL
LIN {X 0,Y 141.504,Z 767.104,A -85,B 0,C 180,E1 6184.916,E2 6184.916} C_VEL
LIN {X 0,Y 148.841,Z 761.12,A -85,B 0,C 180,E1 6177.494,E2 6177.494} C_VEL
LIN {X 0,Y 157.628,Z 753.514,A -85,B 0,C 180,E1 6171.101,E2 6171.101} C_VEL
LIN {X 0,Y 167.373,Z 744.349,A -85,B 0,C 180,E1 6165.66,E2 6165.66} C_VEL
LIN {X 0,Y 177.682,Z 733.655,A -85,B 0,C 180,E1 6161.06,E2 6161.06} C_VEL
LIN {X 0,Y 188.193,Z 721.441,A -85,B 0,C 180,E1 6157.163,E2 6157.163} C_VEL
LIN {X 0,Y 197.936,Z 708.614,A -85,B 0,C 180,E1 6154.064,E2 6154.064} C_VEL
LIN {X 0,Y 207.38,Z 694.44,A -85,B 0,C 180,E1 6151.421,E2 6151.421} C_VEL
LIN {X 0,Y 216.376,Z 678.763,A -85,B 0,C 180,E1 6149.152,E2 6149.152} C_VEL
LIN {X 0,Y 224.431,Z 662.127,A -85,B 0,C 180,E1 6147.282,E2 6147.282} C_VEL
LIN {X 0,Y 231.427,Z 644.54,A -85,B 0,C 180,E1 6145.739,E2 6145.739} C_VEL
LIN {X 0,Y 237.288,Z 625.857,A -85,B 0,C 180,E1 6144.477,E2 6144.477} C_VEL
LIN {X 0,Y 241.784,Z 606.454,A -85,B 0,C 180,E1 6143.492,E2 6143.492} C_VEL
LIN {X 0,Y 244.786,Z 586.673,A -85,B 0,C 180,E1 6142.769,E2 6142.769} C_VEL
LIN {X 0,Y 250.009,Z 532.343,A -85,B 0,C 180,E1 6141.543,E2 6141.543} C_VEL
LIN {X 0,Y 254.254,Z 488.678,A -85,B 0,C 180,E1 6140.65,E2 6140.65} C_VEL
LIN {X 0,Y 250.937,Z 481.573,A -85,B 0,C 180,E1 6137.269,E2 6137.269} C_VEL
LIN {X 0,Y 248.614,Z 477.126,A -85,B 0,C 180,E1 6134.32,E2 6134.32} C_VEL
LIN {X 0,Y 247.259,Z 474.553,A -85,B 0,C 180,E1 6132.139,E2 6132.139} C_VEL
LIN {X 0,Y 245.584,Z 471.298,A -85,B 0,C 180,E1 6128.193,E2 6128.193} C_VEL
LIN {X 0,Y 244.724,Z 470.833,A -85,B 0,C 180,E1 6122.811,E2 6122.811} C_VEL
LIN {X 0,Y 245.064,Z 471.614,A -85,B 0,C 180,E1 6119.767,E2 6119.767} C_VEL
LIN {X 0,Y 246.412,Z 475.312,A -85,B 0,C 180,E1 6115.462,E2 6115.462} C_VEL
LIN {X 0,Y 248.546,Z 480.442,A -85,B 0,C 180,E1 6111.674,E2 6111.674} C_VEL
LIN {X 0,Y 251.166,Z 487.048,A -85,B 0,C 180,E1 6108.287,E2 6108.287} C_VEL
LIN {X 0,Y 254.131,Z 494.822,A -85,B 0,C 180,E1 6105.227,E2 6105.227} C_VEL
LIN {X 0,Y 242.245,Z 609.222,A -85,B 0,C 180,E1 6102.786,E2 6102.786} C_VEL
LIN {X 0,Y 238.249,Z 630.425,A -85,B 0,C 180,E1 6102.145,E2 6102.145} C_VEL
LIN {X 0,Y 234.022,Z 646.228,A -85,B 0,C 180,E1 6101.524,E2 6101.524} C_VEL
LIN {X 0,Y 231.339,Z 653.581,A -85,B 0,C 180,E1 6101.417,E2 6101.417} C_VEL
LIN {X 0,Y 222.223,Z 671.527,A -85,B 0,C 180,E1 6101.838,E2 6101.838} C_VEL
LIN {X 0,Y 218.865,Z 678.321,A -85,B 0,C 180,E1 6101.637,E2 6101.637} C_VEL
LIN {X 0,Y 209.474,Z 697.227,A -85,B 0,C 180,E1 6100.1,E2 6100.1} C_VEL
LIN {X 0,Y 199.274,Z 714.635,A -85,B 0,C 180,E1 6098.157,E2 6098.157} C_VEL
LIN {X 0,Y 188.2,Z 731.072,A -85,B 0,C 180,E1 6095.659,E2 6095.659} C_VEL
LIN {X 0,Y 176.835,Z 745.991,A -85,B 0,C 180,E1 6092.583,E2 6092.583} C_VEL
LIN {X 0,Y 165.767,Z 759.117,A -85,B 0,C 180,E1 6088.923,E2 6088.923} C_VEL
LIN {X 0,Y 154.275,Z 771.737,A -85,B 0,C 180,E1 6084.106,E2 6084.106} C_VEL
LIN {X 0,Y 143.565,Z 782.883,A -85,B 0,C 180,E1 6078.174,E2 6078.174} C_VEL
LIN {X 0,Y 134.267,Z 792.519,A -85,B 0,C 180,E1 6070.942,E2 6070.942} C_VEL
LIN {X 0,Y 127.095,Z 800.561,A -85,B 0,C 180,E1 6062.34,E2 6062.34} C_VEL
LIN {X 0,Y 122.95,Z 806.617,A -85,B 0,C 180,E1 6052.975,E2 6052.975} C_VEL
LIN {X 0,Y 121.864,Z 810.769,A -85,B 0,C 180,E1 6043.281,E2 6043.281} C_VEL
LIN {X 0,Y 122.895,Z 812.832,A -85,B 0,C 180,E1 6035.134,E2 6035.134} C_VEL
LIN {X 0,Y 123.784,Z 813.301,A -85,B 0,C 180,E1 6030,E2 6030} C_VEL
LIN {X 0,Y 122.896,Z 812.82,A -85,B 0,C 180,E1 6024.866,E2 6024.866} C_VEL
LIN {X 0,Y 121.864,Z 810.745,A -85,B 0,C 180,E1 6016.719,E2 6016.719} C_VEL
LIN {X 0,Y 122.954,Z 806.574,A -85,B 0,C 180,E1 6007.025,E2 6007.025} C_VEL
LIN {X 0,Y 127.094,Z 800.499,A -85,B 0,C 180,E1 5997.66,E2 5997.66} C_VEL
LIN {X 0,Y 134.264,Z 792.434,A -85,B 0,C 180,E1 5989.057,E2 5989.057} C_VEL
LIN {X 0,Y 143.56,Z 782.769,A -85,B 0,C 180,E1 5981.823,E2 5981.823} C_VEL
LIN {X 0,Y 154.269,Z 771.592,A -85,B 0,C 180,E1 5975.891,E2 5975.891} C_VEL
LIN {X 0,Y 165.761,Z 758.938,A -85,B 0,C 180,E1 5971.073,E2 5971.073} C_VEL
LIN {X 0,Y 177.211,Z 745.277,A -85,B 0,C 180,E1 5967.295,E2 5967.295} C_VEL
LIN {X 0,Y 188.593,Z 730.225,A -85,B 0,C 180,E1 5964.236,E2 5964.236} C_VEL
LIN {X 0,Y 199.265,Z 714.311,A -85,B 0,C 180,E1 5961.836,E2 5961.836} C_VEL
LIN {X 0,Y 209.465,Z 696.83,A -85,B 0,C 180,E1 5959.893,E2 5959.893} C_VEL
LIN {X 0,Y 218.586,Z 678.45,A -85,B 0,C 180,E1 5958.398,E2 5958.398} C_VEL
LIN {X 0,Y 226.645,Z 658.732,A -85,B 0,C 180,E1 5957.239,E2 5957.239} C_VEL
LIN {X 0,Y 233.138,Z 638.339,A -85,B 0,C 180,E1 5956.348,E2 5956.348} C_VEL
LIN {X 0,Y 237.892,Z 617.644,A -85,B 0,C 180,E1 5955.666,E2 5955.666} C_VEL
LIN {X 0,Y 240.959,Z 596.18,A -85,B 0,C 180,E1 5955.137,E2 5955.137} C_VEL
LIN {X 0,Y 251.058,Z 499.141,A -85,B 0,C 180,E1 5953.12,E2 5953.12} C_VEL
LIN {X 0,Y 248.131,Z 491.094,A -85,B 0,C 180,E1 5949.626,E2 5949.626} C_VEL
LIN {X 0,Y 245.995,Z 485.503,A -85,B 0,C 180,E1 5946.3,E2 5946.3} C_VEL
LIN {X 0,Y 244.629,Z 481.893,A -85,B 0,C 180,E1 5943.28,E2 5943.28} C_VEL
LIN {X 0,Y 243.681,Z 479.016,A -85,B 0,C 180,E1 5939.529,E2 5939.529} C_VEL
LIN {X 0,Y 243.628,Z 478.519,A -85,B 0,C 180,E1 5934.583,E2 5934.583} C_VEL
LIN {X 0,Y 244.54,Z 479.475,A -85,B 0,C 180,E1 5931.061,E2 5931.061} C_VEL
LIN {X 0,Y 246.505,Z 483.434,A -85,B 0,C 180,E1 5926.871,E2 5926.871} C_VEL
LIN {X 0,Y 248.58,Z 487.711,A -85,B 0,C 180,E1 5923.886,E2 5923.886} C_VEL
LIN {X 0,Y 251.249,Z 493.513,A -85,B 0,C 180,E1 5920.869,E2 5920.869} C_VEL
LIN {X 0,Y 242.355,Z 583.135,A -85,B 0,C 180,E1 5919.011,E2 5919.011} C_VEL
LIN {X 0,Y 239.66,Z 602.702,A -85,B 0,C 180,E1 5918.364,E2 5918.364} C_VEL
LIN {X 0,Y 235.43,Z 622.086,A -85,B 0,C 180,E1 5917.471,E2 5917.471} C_VEL
LIN {X 0,Y 229.813,Z 640.766,A -85,B 0,C 180,E1 5916.32,E2 5916.32} C_VEL
LIN {X 0,Y 222.797,Z 658.922,A -85,B 0,C 180,E1 5914.859,E2 5914.859} C_VEL
LIN {X 0,Y 214.306,Z 676.668,A -85,B 0,C 180,E1 5913.011,E2 5913.011} C_VEL
LIN {X 0,Y 204.999,Z 692.902,A -85,B 0,C 180,E1 5910.807,E2 5910.807} C_VEL
LIN {X 0,Y 194.828,Z 707.997,A -85,B 0,C 180,E1 5908.138,E2 5908.138} C_VEL
LIN {X 0,Y 184.325,Z 721.512,A -85,B 0,C 180,E1 5904.992,E2 5904.992} C_VEL
LIN {X 0,Y 173.339,Z 733.908,A -85,B 0,C 180,E1 5901.14,E2 5901.14} C_VEL
LIN {X 0,Y 162.495,Z 744.757,A -85,B 0,C 180,E1 5896.557,E2 5896.557} C_VEL
LIN {X 0,Y 152.151,Z 754.071,A -85,B 0,C 180,E1 5891.081,E2 5891.081} C_VEL
LIN {X 0,Y 142.731,Z 761.826,A -85,B 0,C 180,E1 5884.569,E2 5884.569} C_VEL
LIN {X 0,Y 134.757,Z 767.961,A -85,B 0,C 180,E1 5876.91,E2 5876.91} C_VEL
LIN {X 0,Y 129.039,Z 772.197,A -85,B 0,C 180,E1 5868.523,E2 5868.523} C_VEL
LIN {X 0,Y 125.521,Z 774.784,A -85,B 0,C 180,E1 5859.167,E2 5859.167} C_VEL
LIN {X 0,Y 124.474,Z 775.588,A -85,B 0,C 180,E1 5850,E2 5850} C_VEL
LIN {X 0,Y 125.504,Z 774.814,A -85,B 0,C 180,E1 5840.832,E2 5840.832} C_VEL
LIN {X 0,Y 128.775,Z 772.422,A -85,B 0,C 180,E1 5831.907,E2 5831.907} C_VEL
LIN {X 0,Y 134.36,Z 768.308,A -85,B 0,C 180,E1 5823.482,E2 5823.482} C_VEL
LIN {X 0,Y 141.767,Z 762.656,A -85,B 0,C 180,E1 5816.141,E2 5816.141} C_VEL
LIN {X 0,Y 151.002,Z 755.155,A -85,B 0,C 180,E1 5809.542,E2 5809.542} C_VEL
LIN {X 0,Y 161.192,Z 746.108,A -85,B 0,C 180,E1 5803.986,E2 5803.986} C_VEL
LIN {X 0,Y 171.921,Z 735.549,A -85,B 0,C 180,E1 5799.333,E2 5799.333} C_VEL
LIN {X 0,Y 182.816,Z 723.493,A -85,B 0,C 180,E1 5795.424,E2 5795.424} C_VEL
LIN {X 0,Y 193.535,Z 709.99,A -85,B 0,C 180,E1 5792.15,E2 5792.15} C_VEL
LIN {X 0,Y 203.376,Z 695.74,A -85,B 0,C 180,E1 5789.523,E2 5789.523} C_VEL
LIN {X 0,Y 212.646,Z 680.114,A -85,B 0,C 180,E1 5787.296,E2 5787.296} C_VEL
LIN {X 0,Y 221.33,Z 662.676,A -85,B 0,C 180,E1 5785.382,E2 5785.382} C_VEL
LIN {X 0,Y 228.522,Z 644.98,A -85,B 0,C 180,E1 5783.877,E2 5783.877} C_VEL
LIN {X 0,Y 234.545,Z 626.145,A -85,B 0,C 180,E1 5782.645,E2 5782.645} C_VEL
LIN {X 0,Y 239.215,Z 606.245,A -85,B 0,C 180,E1 5781.672,E2 5781.672} C_VEL
LIN {X 0,Y 242.276,Z 586.007,A -85,B 0,C 180,E1 5780.962,E2 5780.962} C_VEL
LIN {X 0,Y 248.182,Z 526.446,A -85,B 0,C 180,E1 5779.669,E2 5779.669} C_VEL
LIN {X 0,Y 251.482,Z 493.706,A -85,B 0,C 180,E1 5779.028,E2 5779.028} C_VEL
LIN {X 0,Y 248.636,Z 487.499,A -85,B 0,C 180,E1 5775.751,E2 5775.751} C_VEL
LIN {X 0,Y 246.304,Z 482.635,A -85,B 0,C 180,E1 5772.187,E2 5772.187} C_VEL
LIN {X 0,Y 244.548,Z 479.2,A -85,B 0,C 180,E1 5767.991,E2 5767.991} C_VEL
LIN {X 0,Y 243.742,Z 478.774,A -85,B 0,C 180,E1 5762.822,E2 5762.822} C_VEL
LIN {X 0,Y 244.03,Z 479.5,A -85,B 0,C 180,E1 5760,E2 5760} C_VEL
LIN {X 0,Y 245.205,Z 482.992,A -85,B 0,C 180,E1 5755.908,E2 5755.908} C_VEL
LIN {X 0,Y 247.12,Z 487.976,A -85,B 0,C 180,E1 5752.211,E2 5752.211} C_VEL
LIN {X 0,Y 249.46,Z 494.293,A -85,B 0,C 180,E1 5748.967,E2 5748.967} C_VEL
LIN {X 0,Y 251.264,Z 499.644,A -85,B 0,C 180,E1 5746.863,E2 5746.863} C_VEL
LIN {X 0,Y 239.688,Z 608.346,A -85,B 0,C 180,E1 5744.603,E2 5744.603} C_VEL
LIN {X 0,Y 235.654,Z 629.381,A -85,B 0,C 180,E1 5743.991,E2 5743.991} C_VEL
LIN {X 0,Y 230.013,Z 649.616,A -85,B 0,C 180,E1 5743.214,E2 5743.214} C_VEL
LIN {X 0,Y 222.632,Z 669.643,A -85,B 0,C 180,E1 5742.191,E2 5742.191} C_VEL
LIN {X 0,Y 218.865,Z 678.321,A -85,B 0,C 180,E1 5741.637,E2 5741.637} C_VEL
LIN {X 0,Y 215.317,Z 685.172,A -85,B 0,C 180,E1 5741.39,E2 5741.39} C_VEL
LIN {X 0,Y 204.558,Z 700.844,A -85,B 0,C 180,E1 5741.432,E2 5741.432} C_VEL
LIN {X 0,Y 200.213,Z 707.158,A -85,B 0,C 180,E1 5741.081,E2 5741.081} C_VEL
LIN {X 0,Y 199.642,Z 708.04,A -85,B 0,C 180,E1 5740.987,E2 5740.987} C_VEL
LIN {X 0,Y 189.376,Z 723.627,A -85,B 0,C 180,E1 5738.96,E2 5738.96} C_VEL
LIN {X 0,Y 177.583,Z 739.321,A -85,B 0,C 180,E1 5736.193,E2 5736.193} C_VEL
LIN {X 0,Y 165.116,Z 754.037,A -85,B 0,C 180,E1 5732.6,E2 5732.6} C_VEL
LIN {X 0,Y 152.981,Z 767.021,A -85,B 0,C 180,E1 5728.171,E2 5728.171} C_VEL
LIN {X 0,Y 141.012,Z 778.903,A -85,B 0,C 180,E1 5722.427,E2 5722.427} C_VEL
LIN {X 0,Y 130.5,Z 788.962,A -85,B 0,C 180,E1 5715.44,E2 5715.44} C_VEL
LIN {X 0,Y 121.838,Z 797.526,A -85,B 0,C 180,E1 5706.802,E2 5706.802} C_VEL
LIN {X 0,Y 116.251,Z 804.077,A -85,B 0,C 180,E1 5697.118,E2 5697.118} C_VEL
LIN {X 0,Y 113.97,Z 808.695,A -85,B 0,C 180,E1 5686.828,E2 5686.828} C_VEL
LIN {X 0,Y 114.5,Z 811.206,A -85,B 0,C 180,E1 5677.526,E2 5677.526} C_VEL
LIN {X 0,Y 115.769,Z 812.044,A -85,B 0,C 180,E1 5670.99,E2 5670.99} C_VEL
LIN {X 0,Y 115.497,Z 811.914,A -85,B 0,C 180,E1 5667.519,E2 5667.519} C_VEL
LIN {X 0,Y 114.081,Z 810.561,A -85,B 0,C 180,E1 5659.394,E2 5659.394} C_VEL
LIN {X 0,Y 114.391,Z 807.231,A -85,B 0,C 180,E1 5649.536,E2 5649.536} C_VEL
LIN {X 0,Y 117.589,Z 802.212,A -85,B 0,C 180,E1 5639.89,E2 5639.89} C_VEL
LIN {X 0,Y 124.135,Z 795.049,A -85,B 0,C 180,E1 5630.484,E2 5630.484} C_VEL
LIN {X 0,Y 133.222,Z 786.193,A -85,B 0,C 180,E1 5622.489,E2 5622.489} C_VEL
LIN {X 0,Y 144.278,Z 775.535,A -85,B 0,C 180,E1 5615.826,E2 5615.826} C_VEL
LIN {X 0,Y 155.791,Z 763.869,A -85,B 0,C 180,E1 5610.686,E2 5610.686} C_VEL
LIN {X 0,Y 167.847,Z 750.69,A -85,B 0,C 180,E1 5606.536,E2 5606.536} C_VEL
LIN {X 0,Y 179.659,Z 736.401,A -85,B 0,C 180,E1 5603.274,E2 5603.274} C_VEL
LIN {X 0,Y 190.819,Z 721.24,A -85,B 0,C 180,E1 5600.726,E2 5600.726} C_VEL
LIN {X 0,Y 201.564,Z 704.565,A -85,B 0,C 180,E1 5598.661,E2 5598.661} C_VEL
LIN {X 0,Y 211.361,Z 686.846,A -85,B 0,C 180,E1 5597.055,E2 5597.055} C_VEL
LIN {X 0,Y 220.062,Z 668.056,A -85,B 0,C 180,E1 5595.819,E2 5595.819} C_VEL
LIN {X 0,Y 227.565,Z 647.862,A -85,B 0,C 180,E1 5594.852,E2 5594.852} C_VEL
LIN {X 0,Y 233.312,Z 627.289,A -85,B 0,C 180,E1 5594.109,E2 5594.109} C_VEL
LIN {X 0,Y 237.313,Z 606.212,A -85,B 0,C 180,E1 5593.531,E2 5593.531} C_VEL
LIN {X 0,Y 248.415,Z 503.894,A -85,B 0,C 180,E1 5591.452,E2 5591.452} C_VEL
LIN {X 0,Y 246.22,Z 497.525,A -85,B 0,C 180,E1 5588.465,E2 5588.465} C_VEL
LIN {X 0,Y 244.596,Z 492.903,A -85,B 0,C 180,E1 5585.63,E2 5585.63} C_VEL
LIN {X 0,Y 243.455,Z 489.593,A -85,B 0,C 180,E1 5582.824,E2 5582.824} C_VEL
LIN {X 0,Y 242.665,Z 486.908,A -85,B 0,C 180,E1 5579.291,E2 5579.291} C_VEL
LIN {X 0,Y 242.657,Z 486.463,A -85,B 0,C 180,E1 5574.561,E2 5574.561} C_VEL
LIN {X 0,Y 243.447,Z 487.289,A -85,B 0,C 180,E1 5571.378,E2 5571.378} C_VEL
LIN {X 0,Y 245.246,Z 491.15,A -85,B 0,C 180,E1 5567.281,E2 5567.281} C_VEL
LIN {X 0,Y 247.287,Z 495.563,A -85,B 0,C 180,E1 5564.213,E2 5564.213} C_VEL
LIN {X 0,Y 248.611,Z 498.871,A -85,B 0,C 180,E1 5562.538,E2 5562.538} C_VEL
LIN {X 0,Y 239.939,Z 583.793,A -85,B 0,C 180,E1 5560.816,E2 5560.816} C_VEL
LIN {X 0,Y 237.164,Z 603.419,A -85,B 0,C 180,E1 5560.183,E2 5560.183} C_VEL
LIN {X 0,Y 232.949,Z 622.393,A -85,B 0,C 180,E1 5559.337,E2 5559.337} C_VEL
LIN {X 0,Y 227.183,Z 641.204,A -85,B 0,C 180,E1 5558.219,E2 5558.219} C_VEL
LIN {X 0,Y 219.793,Z 659.877,A -85,B 0,C 180,E1 5556.764,E2 5556.764} C_VEL
LIN {X 0,Y 211.251,Z 677.308,A -85,B 0,C 180,E1 5555.006,E2 5555.006} C_VEL
LIN {X 0,Y 201.648,Z 693.632,A -85,B 0,C 180,E1 5552.859,E2 5552.859} C_VEL
LIN {X 0,Y 191.16,Z 708.768,A -85,B 0,C 180,E1 5550.254,E2 5550.254} C_VEL
LIN {X 0,Y 179.903,Z 722.764,A -85,B 0,C 180,E1 5547.055,E2 5547.055} C_VEL
LIN {X 0,Y 168.485,Z 735.143,A -85,B 0,C 180,E1 5543.237,E2 5543.237} C_VEL
LIN {X 0,Y 157.151,Z 745.983,A -85,B 0,C 180,E1 5538.655,E2 5538.655} C_VEL
LIN {X 0,Y 146.265,Z 755.289,A -85,B 0,C 180,E1 5533.124,E2 5533.124} C_VEL
LIN {X 0,Y 136.273,Z 763.038,A -85,B 0,C 180,E1 5526.462,E2 5526.462} C_VEL
LIN {X 0,Y 127.733,Z 769.169,A -85,B 0,C 180,E1 5518.521,E2 5518.521} C_VEL
LIN {X 0,Y 121.549,Z 773.402,A -85,B 0,C 180,E1 5509.71,E2 5509.71} C_VEL
LIN {X 0,Y 117.713,Z 775.986,A -85,B 0,C 180,E1 5499.781,E2 5499.781} C_VEL
LIN {X 0,Y 116.565,Z 776.79,A -85,B 0,C 180,E1 5490,E2 5490} C_VEL
LIN {X 0,Y 117.695,Z 776.016,A -85,B 0,C 180,E1 5480.218,E2 5480.218} C_VEL
LIN {X 0,Y 121.265,Z 773.625,A -85,B 0,C 180,E1 5470.743,E2 5470.743} C_VEL
LIN {X 0,Y 127.31,Z 769.512,A -85,B 0,C 180,E1 5461.887,E2 5461.887} C_VEL
LIN {X 0,Y 135.25,Z 763.862,A -85,B 0,C 180,E1 5454.267,E2 5454.267} C_VEL
LIN {X 0,Y 145.057,Z 756.365,A -85,B 0,C 180,E1 5447.509,E2 5447.509} C_VEL
LIN {X 0,Y 155.792,Z 747.325,A -85,B 0,C 180,E1 5441.888,E2 5441.888} C_VEL
LIN {X 0,Y 167.014,Z 736.776,A -85,B 0,C 180,E1 5437.231,E2 5437.231} C_VEL
LIN {X 0,Y 178.346,Z 724.735,A -85,B 0,C 180,E1 5433.352,E2 5433.352} C_VEL
LIN {X 0,Y 188.773,Z 712.122,A -85,B 0,C 180,E1 5430.308,E2 5430.308} C_VEL
LIN {X 0,Y 199.605,Z 697.039,A -85,B 0,C 180,E1 5427.551,E2 5427.551} C_VEL
LIN {X 0,Y 209.36,Z 681.087,A -85,B 0,C 180,E1 5425.33,E2 5425.33} C_VEL
LIN {X 0,Y 218.091,Z 664.058,A -85,B 0,C 180,E1 5423.508,E2 5423.508} C_VEL
LIN {X 0,Y 225.453,Z 646.525,A -85,B 0,C 180,E1 5422.049,E2 5422.049} C_VEL
LIN {X 0,Y 231.634,Z 627.886,A -85,B 0,C 180,E1 5420.852,E2 5420.852} C_VEL
LIN {X 0,Y 236.407,Z 608.474,A -85,B 0,C 180,E1 5419.912,E2 5419.912} C_VEL
LIN {X 0,Y 239.62,Z 588.738,A -85,B 0,C 180,E1 5419.214,E2 5419.214} C_VEL
LIN {X 0,Y 244.839,Z 537.832,A -85,B 0,C 180,E1 5418.097,E2 5418.097} C_VEL
LIN {X 0,Y 248.836,Z 498.724,A -85,B 0,C 180,E1 5417.299,E2 5417.299} C_VEL
LIN {X 0,Y 246.359,Z 493.117,A -85,B 0,C 180,E1 5413.975,E2 5413.975} C_VEL
LIN {X 0,Y 244.838,Z 489.99,A -85,B 0,C 180,E1 5411.305,E2 5411.305} C_VEL
LIN {X 0,Y 243.503,Z 487.102,A -85,B 0,C 180,E1 5407.788,E2 5407.788} C_VEL
LIN {X 0,Y 242.773,Z 486.747,A -85,B 0,C 180,E1 5402.597,E2 5402.597} C_VEL
LIN {X 0,Y 243.007,Z 487.386,A -85,B 0,C 180,E1 5400.236,E2 5400.236} C_VEL
LIN {X 0,Y 244.049,Z 490.824,A -85,B 0,C 180,E1 5396.242,E2 5396.242} C_VEL
LIN {X 0,Y 245.714,Z 495.533,A -85,B 0,C 180,E1 5392.754,E2 5392.754} C_VEL
LIN {X 0,Y 247.827,Z 501.665,A -85,B 0,C 180,E1 5389.599,E2 5389.599} C_VEL
LIN {X 0,Y 248.637,Z 504.328,A -85,B 0,C 180,E1 5388.54,E2 5388.54} C_VEL
LIN {X 0,Y 237.373,Z 607.494,A -85,B 0,C 180,E1 5386.457,E2 5386.457} C_VEL
LIN {X 0,Y 233.244,Z 628.586,A -85,B 0,C 180,E1 5385.869,E2 5385.869} C_VEL
LIN {X 0,Y 227.574,Z 648.582,A -85,B 0,C 180,E1 5385.139,E2 5385.139} C_VEL
LIN {X 0,Y 220.187,Z 668.326,A -85,B 0,C 180,E1 5384.19,E2 5384.19} C_VEL
LIN {X 0,Y 211.279,Z 687.467,A -85,B 0,C 180,E1 5382.924,E2 5382.924} C_VEL
LIN {X 0,Y 201.137,Z 705.669,A -85,B 0,C 180,E1 5381.254,E2 5381.254} C_VEL
LIN {X 0,Y 199.642,Z 708.04,A -85,B 0,C 180,E1 5380.987,E2 5380.987} C_VEL
LIN {X 0,Y 195.24,Z 714.33,A -85,B 0,C 180,E1 5380.507,E2 5380.507} C_VEL
LIN {X 0,Y 181.875,Z 729.241,A -85,B 0,C 180,E1 5379.977,E2 5379.977} C_VEL
LIN {X 0,Y 177.003,Z 734.779,A -85,B 0,C 180,E1 5379.281,E2 5379.281} C_VEL
LIN {X 0,Y 164.973,Z 748.868,A -85,B 0,C 180,E1 5376.226,E2 5376.226} C_VEL
LIN {X 0,Y 152.301,Z 762.168,A -85,B 0,C 180,E1 5372.218,E2 5372.218} C_VEL
LIN {X 0,Y 139.57,Z 774.389,A -85,B 0,C 180,E1 5366.945,E2 5366.945} C_VEL
LIN {X 0,Y 127.589,Z 785.152,A -85,B 0,C 180,E1 5360.171,E2 5360.171} C_VEL
LIN {X 0,Y 117.375,Z 794.256,A -85,B 0,C 180,E1 5351.638,E2 5351.638} C_VEL
LIN {X 0,Y 110.187,Z 801.303,A -85,B 0,C 180,E1 5341.755,E2 5341.755} C_VEL
LIN {X 0,Y 106.474,Z 806.421,A -85,B 0,C 180,E1 5330.906,E2 5330.906} C_VEL
LIN {X 0,Y 106.167,Z 809.553,A -85,B 0,C 180,E1 5320.307,E2 5320.307} C_VEL
LIN {X 0,Y 107.607,Z 810.749,A -85,B 0,C 180,E1 5312.13,E2 5312.13} C_VEL
LIN {X 0,Y 107.895,Z 810.868,A -85,B 0,C 180,E1 5309.469,E2 5309.469} C_VEL
LIN {X 0,Y 106.454,Z 809.957,A -85,B 0,C 180,E1 5301.901,E2 5301.901} C_VEL
LIN {X 0,Y 106.107,Z 807.406,A -85,B 0,C 180,E1 5291.883,E2 5291.883} C_VEL
LIN {X 0,Y 108.924,Z 802.762,A -85,B 0,C 180,E1 5280.889,E2 5280.889} C_VEL
LIN {X 0,Y 115.268,Z 796.19,A -85,B 0,C 180,E1 5270.713,E2 5270.713} C_VEL
LIN {X 0,Y 124.779,Z 787.589,A -85,B 0,C 180,E1 5261.825,E2 5261.825} C_VEL
LIN {X 0,Y 136.227,Z 777.367,A -85,B 0,C 180,E1 5254.713,E2 5254.713} C_VEL
LIN {X 0,Y 148.753,Z 765.575,A -85,B 0,C 180,E1 5249.099,E2 5249.099} C_VEL
LIN {X 0,Y 161.767,Z 752.23,A -85,B 0,C 180,E1 5244.693,E2 5244.693} C_VEL
LIN {X 0,Y 174.408,Z 737.778,A -85,B 0,C 180,E1 5241.32,E2 5241.32} C_VEL
LIN {X 0,Y 186.765,Z 721.753,A -85,B 0,C 180,E1 5238.638,E2 5238.638} C_VEL
LIN {X 0,Y 198.205,Z 704.643,A -85,B 0,C 180,E1 5236.576,E2 5236.576} C_VEL
LIN {X 0,Y 208.478,Z 686.612,A -85,B 0,C 180,E1 5235.009,E2 5235.009} C_VEL
LIN {X 0,Y 217.744,Z 667.053,A -85,B 0,C 180,E1 5233.795,E2 5233.795} C_VEL
LIN {X 0,Y 225.4,Z 646.768,A -85,B 0,C 180,E1 5232.886,E2 5232.886} C_VEL
LIN {X 0,Y 231.205,Z 626.288,A -85,B 0,C 180,E1 5232.189,E2 5232.189} C_VEL
LIN {X 0,Y 235.253,Z 605.32,A -85,B 0,C 180,E1 5231.642,E2 5231.642} C_VEL
LIN {X 0,Y 245.951,Z 508.72,A -85,B 0,C 180,E1 5229.712,E2 5229.712} C_VEL
LIN {X 0,Y 244.101,Z 502.858,A -85,B 0,C 180,E1 5226.703,E2 5226.703} C_VEL
LIN {X 0,Y 242.489,Z 497.782,A -85,B 0,C 180,E1 5222.954,E2 5222.954} C_VEL
LIN {X 0,Y 241.653,Z 494.801,A -85,B 0,C 180,E1 5219.051,E2 5219.051} C_VEL
LIN {X 0,Y 241.686,Z 494.409,A -85,B 0,C 180,E1 5214.539,E2 5214.539} C_VEL
LIN {X 0,Y 242.394,Z 495.209,A -85,B 0,C 180,E1 5211.579,E2 5211.579} C_VEL
LIN {X 0,Y 244.01,Z 498.865,A -85,B 0,C 180,E1 5207.697,E2 5207.697} C_VEL
LIN {X 0,Y 246.034,Z 503.479,A -85,B 0,C 180,E1 5204.502,E2 5204.502} C_VEL
LIN {X 0,Y 246.186,Z 504.23,A -85,B 0,C 180,E1 5204.243,E2 5204.243} C_VEL
LIN {X 0,Y 237.734,Z 584.723,A -85,B 0,C 180,E1 5202.649,E2 5202.649} C_VEL
LIN {X 0,Y 234.859,Z 604.39,A -85,B 0,C 180,E1 5202.028,E2 5202.028} C_VEL
LIN {X 0,Y 230.507,Z 623.429,A -85,B 0,C 180,E1 5201.203,E2 5201.203} C_VEL
LIN {X 0,Y 224.806,Z 641.606,A -85,B 0,C 180,E1 5200.161,E2 5200.161} C_VEL
LIN {X 0,Y 217.408,Z 659.997,A -85,B 0,C 180,E1 5198.79,E2 5198.79} C_VEL
LIN {X 0,Y 208.871,Z 677.148,A -85,B 0,C 180,E1 5197.141,E2 5197.141} C_VEL
LIN {X 0,Y 199.409,Z 693.004,A -85,B 0,C 180,E1 5195.166,E2 5195.166} C_VEL
LIN {X 0,Y 188.947,Z 707.92,A -85,B 0,C 180,E1 5192.746,E2 5192.746} C_VEL
LIN {X 0,Y 178.011,Z 721.363,A -85,B 0,C 180,E1 5189.879,E2 5189.879} C_VEL
LIN {X 0,Y 166.769,Z 733.436,A -85,B 0,C 180,E1 5186.444,E2 5186.444} C_VEL
LIN {X 0,Y 154.73,Z 744.788,A -85,B 0,C 180,E1 5182.03,E2 5182.03} C_VEL
LIN {X 0,Y 143.009,Z 754.559,A -85,B 0,C 180,E1 5176.644,E2 5176.644} C_VEL
LIN {X 0,Y 132.064,Z 762.73,A -85,B 0,C 180,E1 5170.055,E2 5170.055} C_VEL
LIN {X 0,Y 122.886,Z 768.976,A -85,B 0,C 180,E1 5162.479,E2 5162.479} C_VEL
LIN {X 0,Y 115.542,Z 773.666,A -85,B 0,C 180,E1 5153.457,E2 5153.457} C_VEL
LIN {X 0,Y 110.806,Z 776.59,A -85,B 0,C 180,E1 5143.568,E2 5143.568} C_VEL
LIN {X 0,Y 108.761,Z 777.868,A -85,B 0,C 180,E1 5133.162,E2 5133.162} C_VEL
LIN {X 0,Y 109.169,Z 777.64,A -85,B 0,C 180,E1 5123.162,E2 5123.162} C_VEL
LIN {X 0,Y 111.919,Z 775.987,A -85,B 0,C 180,E1 5113.389,E2 5113.389} C_VEL
LIN {X 0,Y 117.435,Z 772.592,A -85,B 0,C 180,E1 5103.722,E2 5103.722} C_VEL
LIN {X 0,Y 125.513,Z 767.375,A -85,B 0,C 180,E1 5095.002,E2 5095.002} C_VEL
LIN {X 0,Y 135.283,Z 760.595,A -85,B 0,C 180,E1 5087.736,E2 5087.736} C_VEL
LIN {X 0,Y 146.709,Z 751.805,A -85,B 0,C 180,E1 5081.44,E2 5081.44} C_VEL
LIN {X 0,Y 158.107,Z 742.009,A -85,B 0,C 180,E1 5076.571,E2 5076.571} C_VEL
LIN {X 0,Y 170.379,Z 730.03,A -85,B 0,C 180,E1 5072.325,E2 5072.325} C_VEL
LIN {X 0,Y 181.794,Z 717.27,A -85,B 0,C 180,E1 5069.018,E2 5069.018} C_VEL
LIN {X 0,Y 193.26,Z 702.447,A -85,B 0,C 180,E1 5066.156,E2 5066.156} C_VEL
LIN {X 0,Y 203.835,Z 686.379,A -85,B 0,C 180,E1 5063.823,E2 5063.823} C_VEL
LIN {X 0,Y 212.963,Z 669.874,A -85,B 0,C 180,E1 5061.993,E2 5061.993} C_VEL
LIN {X 0,Y 221.36,Z 651.372,A -85,B 0,C 180,E1 5060.409,E2 5060.409} C_VEL
LIN {X 0,Y 228.074,Z 632.648,A -85,B 0,C 180,E1 5059.181,E2 5059.181} C_VEL
LIN {X 0,Y 233.423,Z 612.684,A -85,B 0,C 180,E1 5058.192,E2 5058.192} C_VEL
LIN {X 0,Y 237.08,Z 592.394,A -85,B 0,C 180,E1 5057.457,E2 5057.457} C_VEL
LIN {X 0,Y 241.701,Z 549.071,A -85,B 0,C 180,E1 5056.479,E2 5056.479} C_VEL
LIN {X 0,Y 246.448,Z 504.107,A -85,B 0,C 180,E1 5055.61,E2 5055.61} C_VEL
LIN {X 0,Y 244.598,Z 499.812,A -85,B 0,C 180,E1 5052.753,E2 5052.753} C_VEL
LIN {X 0,Y 243.524,Z 497.514,A -85,B 0,C 180,E1 5050.648,E2 5050.648} C_VEL
LIN {X 0,Y 242.461,Z 495.005,A -85,B 0,C 180,E1 5047.583,E2 5047.583} C_VEL
LIN {X 0,Y 241.799,Z 494.691,A -85,B 0,C 180,E1 5042.608,E2 5042.608} C_VEL
LIN {X 0,Y 242.015,Z 495.465,A -85,B 0,C 180,E1 5040.237,E2 5040.237} C_VEL
LIN {X 0,Y 242.9,Z 498.654,A -85,B 0,C 180,E1 5036.579,E2 5036.579} C_VEL
LIN {X 0,Y 244.31,Z 502.981,A -85,B 0,C 180,E1 5033.361,E2 5033.361} C_VEL
LIN {X 0,Y 246.184,Z 508.907,A -85,B 0,C 180,E1 5030.297,E2 5030.297} C_VEL
LIN {X 0,Y 235.312,Z 606.641,A -85,B 0,C 180,E1 5028.345,E2 5028.345} C_VEL
LIN {X 0,Y 231.103,Z 627.741,A -85,B 0,C 180,E1 5027.785,E2 5027.785} C_VEL
LIN {X 0,Y 225.335,Z 647.729,A -85,B 0,C 180,E1 5027.097,E2 5027.097} C_VEL
LIN {X 0,Y 217.878,Z 667.319,A -85,B 0,C 180,E1 5026.214,E2 5026.214} C_VEL
LIN {X 0,Y 209.031,Z 686.009,A -85,B 0,C 180,E1 5025.061,E2 5025.061} C_VEL
LIN {X 0,Y 198.657,Z 704.279,A -85,B 0,C 180,E1 5023.491,E2 5023.491} C_VEL
LIN {X 0,Y 187.205,Z 721.443,A -85,B 0,C 180,E1 5021.44,E2 5021.44} C_VEL
LIN {X 0,Y 177.003,Z 734.779,A -85,B 0,C 180,E1 5019.281,E2 5019.281} C_VEL
LIN {X 0,Y 172.013,Z 740.25,A -85,B 0,C 180,E1 5018.5,E2 5018.5} C_VEL
LIN {X 0,Y 157.064,Z 753.161,A -85,B 0,C 180,E1 5017.167,E2 5017.167} C_VEL
LIN {X 0,Y 151.738,Z 757.922,A -85,B 0,C 180,E1 5016.048,E2 5016.048} C_VEL
LIN {X 0,Y 138.112,Z 770.609,A -85,B 0,C 180,E1 5011.157,E2 5011.157} C_VEL
LIN {X 0,Y 125.393,Z 781.479,A -85,B 0,C 180,E1 5004.963,E2 5004.963} C_VEL
LIN {X 0,Y 113.8,Z 790.964,A -85,B 0,C 180,E1 4996.821,E2 4996.821} C_VEL
LIN {X 0,Y 104.747,Z 798.638,A -85,B 0,C 180,E1 4986.698,E2 4986.698} C_VEL
LIN {X 0,Y 99.357,Z 804.341,A -85,B 0,C 180,E1 4975.002,E2 4975.002} C_VEL
LIN {X 0,Y 98.035,Z 807.959,A -85,B 0,C 180,E1 4962.966,E2 4962.966} C_VEL
LIN {X 0,Y 99.472,Z 809.483,A -85,B 0,C 180,E1 4952.881,E2 4952.881} C_VEL
LIN {X 0,Y 99.955,Z 809.662,A -85,B 0,C 180,E1 4949.427,E2 4949.427} C_VEL
LIN {X 0,Y 98.402,Z 808.721,A -85,B 0,C 180,E1 4941.233,E2 4941.233} C_VEL
LIN {X 0,Y 98.378,Z 805.947,A -85,B 0,C 180,E1 4929.785,E2 4929.785} C_VEL
LIN {X 0,Y 101.741,Z 801.496,A -85,B 0,C 180,E1 4918.611,E2 4918.611} C_VEL
LIN {X 0,Y 108.939,Z 794.918,A -85,B 0,C 180,E1 4907.934,E2 4907.934} C_VEL
LIN {X 0,Y 119.373,Z 786.31,A -85,B 0,C 180,E1 4898.836,E2 4898.836} C_VEL
LIN {X 0,Y 131.66,Z 776.083,A -85,B 0,C 180,E1 4891.73,E2 4891.73} C_VEL
LIN {X 0,Y 144.968,Z 764.203,A -85,B 0,C 180,E1 4886.193,E2 4886.193} C_VEL
LIN {X 0,Y 158.486,Z 750.924,A -85,B 0,C 180,E1 4881.972,E2 4881.972} C_VEL
LIN {X 0,Y 171.581,Z 736.457,A -85,B 0,C 180,E1 4878.753,E2 4878.753} C_VEL
LIN {X 0,Y 184.302,Z 720.399,A -85,B 0,C 180,E1 4876.216,E2 4876.216} C_VEL
LIN {X 0,Y 196.026,Z 703.244,A -85,B 0,C 180,E1 4874.282,E2 4874.282} C_VEL
LIN {X 0,Y 206.61,Z 684.97,A -85,B 0,C 180,E1 4872.812,E2 4872.812} C_VEL
LIN {X 0,Y 215.484,Z 666.559,A -85,B 0,C 180,E1 4871.755,E2 4871.755} C_VEL
LIN {X 0,Y 223.249,Z 646.468,A -85,B 0,C 180,E1 4870.911,E2 4870.911} C_VEL
LIN {X 0,Y 229.274,Z 625.681,A -85,B 0,C 180,E1 4870.246,E2 4870.246} C_VEL
LIN {X 0,Y 233.44,Z 604.543,A -85,B 0,C 180,E1 4869.724,E2 4869.724} C_VEL
LIN {X 0,Y 243.717,Z 513.688,A -85,B 0,C 180,E1 4867.958,E2 4867.958} C_VEL
LIN {X 0,Y 242.107,Z 508.248,A -85,B 0,C 180,E1 4864.737,E2 4864.737} C_VEL
LIN {X 0,Y 241.151,Z 504.989,A -85,B 0,C 180,E1 4861.9,E2 4861.9} C_VEL
LIN {X 0,Y 240.632,Z 502.694,A -85,B 0,C 180,E1 4858.809,E2 4858.809} C_VEL
LIN {X 0,Y 240.752,Z 502.382,A -85,B 0,C 180,E1 4854.279,E2 4854.279} C_VEL
LIN {X 0,Y 241.343,Z 503.129,A -85,B 0,C 180,E1 4851.782,E2 4851.782} C_VEL
LIN {X 0,Y 242.787,Z 506.581,A -85,B 0,C 180,E1 4848.117,E2 4848.117} C_VEL
LIN {X 0,Y 243.97,Z 509.678,A -85,B 0,C 180,E1 4845.979,E2 4845.979} C_VEL
LIN {X 0,Y 235.774,Z 585.685,A -85,B 0,C 180,E1 4844.514,E2 4844.514} C_VEL
LIN {X 0,Y 232.802,Z 605.363,A -85,B 0,C 180,E1 4843.908,E2 4843.908} C_VEL
LIN {X 0,Y 228.314,Z 624.463,A -85,B 0,C 180,E1 4843.108,E2 4843.108} C_VEL
LIN {X 0,Y 222.262,Z 643.224,A -85,B 0,C 180,E1 4842.067,E2 4842.067} C_VEL
LIN {X 0,Y 214.501,Z 661.875,A -85,B 0,C 180,E1 4840.716,E2 4840.716} C_VEL
LIN {X 0,Y 205.514,Z 679.31,A -85,B 0,C 180,E1 4839.081,E2 4839.081} C_VEL
LIN {X 0,Y 195.394,Z 695.62,A -85,B 0,C 180,E1 4837.081,E2 4837.081} C_VEL
LIN {X 0,Y 184.049,Z 711.054,A -85,B 0,C 180,E1 4834.584,E2 4834.584} C_VEL
LIN {X 0,Y 171.814,Z 725.261,A -85,B 0,C 180,E1 4831.487,E2 4831.487} C_VEL
LIN {X 0,Y 159.514,Z 737.609,A -85,B 0,C 180,E1 4827.799,E2 4827.799} C_VEL
LIN {X 0,Y 147.058,Z 748.516,A -85,B 0,C 180,E1 4823.249,E2 4823.249} C_VEL
LIN {X 0,Y 134.743,Z 757.997,A -85,B 0,C 180,E1 4817.524,E2 4817.524} C_VEL
LIN {X 0,Y 123.326,Z 765.806,A -85,B 0,C 180,E1 4810.434,E2 4810.434} C_VEL
LIN {X 0,Y 113.613,Z 771.822,A -85,B 0,C 180,E1 4801.872,E2 4801.872} C_VEL
LIN {X 0,Y 106.463,Z 775.965,A -85,B 0,C 180,E1 4792.065,E2 4792.065} C_VEL
LIN {X 0,Y 102.147,Z 778.391,A -85,B 0,C 180,E1 4781.289,E2 4781.289} C_VEL
LIN {X 0,Y 100.746,Z 779.193,A -85,B 0,C 180,E1 4770,E2 4770} C_VEL
LIN {X 0,Y 102.128,Z 778.419,A -85,B 0,C 180,E1 4758.709,E2 4758.709} C_VEL
LIN {X 0,Y 106.426,Z 776.031,A -85,B 0,C 180,E1 4747.927,E2 4747.927} C_VEL
LIN {X 0,Y 113.559,Z 771.921,A -85,B 0,C 180,E1 4738.111,E2 4738.111} C_VEL
LIN {X 0,Y 122.718,Z 766.274,A -85,B 0,C 180,E1 4729.936,E2 4729.936} C_VEL
LIN {X 0,Y 133.787,Z 758.784,A -85,B 0,C 180,E1 4722.914,E2 4722.914} C_VEL
LIN {X 0,Y 145.685,Z 749.755,A -85,B 0,C 180,E1 4717.24,E2 4717.24} C_VEL
LIN {X 0,Y 157.934,Z 739.226,A -85,B 0,C 180,E1 4712.65,E2 4712.65} C_VEL
LIN {X 0,Y 170.16,Z 727.216,A -85,B 0,C 180,E1 4708.896,E2 4708.896} C_VEL
LIN {X 0,Y 182.121,Z 713.67,A -85,B 0,C 180,E1 4705.796,E2 4705.796} C_VEL
LIN {X 0,Y 193.227,Z 699.046,A -85,B 0,C 180,E1 4703.3,E2 4703.3} C_VEL
LIN {X 0,Y 203.313,Z 683.449,A -85,B 0,C 180,E1 4701.267,E2 4701.267} C_VEL
LIN {X 0,Y 212.707,Z 666.077,A -85,B 0,C 180,E1 4699.533,E2 4699.533} C_VEL
LIN {X 0,Y 220.463,Z 648.509,A -85,B 0,C 180,E1 4698.174,E2 4698.174} C_VEL
LIN {X 0,Y 226.951,Z 629.916,A -85,B 0,C 180,E1 4697.062,E2 4697.062} C_VEL
LIN {X 0,Y 231.994,Z 610.495,A -85,B 0,C 180,E1 4696.18,E2 4696.18} C_VEL
LIN {X 0,Y 235.428,Z 590.695,A -85,B 0,C 180,E1 4695.516,E2 4695.516} C_VEL
LIN {X 0,Y 240.775,Z 541.624,A -85,B 0,C 180,E1 4694.485,E2 4694.485} C_VEL
LIN {X 0,Y 244.244,Z 509.703,A -85,B 0,C 180,E1 4693.894,E2 4693.894} C_VEL
LIN {X 0,Y 242.548,Z 505.607,A -85,B 0,C 180,E1 4690.691,E2 4690.691} C_VEL
LIN {X 0,Y 241.356,Z 502.858,A -85,B 0,C 180,E1 4687.14,E2 4687.14} C_VEL
LIN {X 0,Y 240.832,Z 502.679,A -85,B 0,C 180,E1 4682.38,E2 4682.38} C_VEL
LIN {X 0,Y 240.997,Z 503.351,A -85,B 0,C 180,E1 4680.476,E2 4680.476} C_VEL
LIN {X 0,Y 241.725,Z 506.331,A -85,B 0,C 180,E1 4677.037,E2 4677.037} C_VEL
LIN {X 0,Y 242.963,Z 510.535,A -85,B 0,C 180,E1 4673.918,E2 4673.918} C_VEL
LIN {X 0,Y 243.972,Z 514.154,A -85,B 0,C 180,E1 4671.989,E2 4671.989} C_VEL
LIN {X 0,Y 233.511,Z 605.792,A -85,B 0,C 180,E1 4670.264,E2 4670.264} C_VEL
LIN {X 0,Y 229.253,Z 626.792,A -85,B 0,C 180,E1 4669.738,E2 4669.738} C_VEL
LIN {X 0,Y 223.491,Z 646.514,A -85,B 0,C 180,E1 4669.105,E2 4669.105} C_VEL
LIN {X 0,Y 215.959,Z 666.059,A -85,B 0,C 180,E1 4668.29,E2 4668.29} C_VEL
LIN {X 0,Y 206.616,Z 685.431,A -85,B 0,C 180,E1 4667.18,E2 4667.18} C_VEL
LIN {X 0,Y 196.033,Z 703.611,A -85,B 0,C 180,E1 4665.71,E2 4665.71} C_VEL
LIN {X 0,Y 184.308,Z 720.702,A -85,B 0,C 180,E1 4663.777,E2 4663.777} C_VEL
LIN {X 0,Y 171.587,Z 736.704,A -85,B 0,C 180,E1 4661.241,E2 4661.241} C_VEL
LIN {X 0,Y 158.492,Z 751.13,A -85,B 0,C 180,E1 4658.023,E2 4658.023} C_VEL
LIN {X 0,Y 151.738,Z 757.922,A -85,B 0,C 180,E1 4656.048,E2 4656.048} C_VEL
LIN {X 0,Y 146.355,Z 762.485,A -85,B 0,C 180,E1 4654.795,E2 4654.795} C_VEL
LIN {X 0,Y 130.468,Z 773.041,A -85,B 0,C 180,E1 4652.132,E2 4652.132} C_VEL
LIN {X 0,Y 125.033,Z 776.84,A -85,B 0,C 180,E1 4650.328,E2 4650.328} C_VEL
LIN {X 0,Y 113.061,Z 786.062,A -85,B 0,C 180,E1 4643.584,E2 4643.584} C_VEL
LIN {X 0,Y 102.404,Z 794.079,A -85,B 0,C 180,E1 4634.666,E2 4634.666} C_VEL
LIN {X 0,Y 94.429,Z 800.558,A -85,B 0,C 180,E1 4623.407,E2 4623.407} C_VEL
LIN {X 0,Y 90.457,Z 805.134,A -85,B 0,C 180,E1 4610.714,E2 4610.714} C_VEL
LIN {X 0,Y 90.51,Z 807.709,A -85,B 0,C 180,E1 4598.256,E2 4598.256} C_VEL
LIN {X 0,Y 92.096,Z 808.487,A -85,B 0,C 180,E1 4590,E2 4590} C_VEL
LIN {X 0,Y 90.353,Z 807.482,A -85,B 0,C 180,E1 4580.445,E2 4580.445} C_VEL
LIN {X 0,Y 90.668,Z 804.69,A -85,B 0,C 180,E1 4567.98,E2 4567.98} C_VEL
LIN {X 0,Y 94.735,Z 800.228,A -85,B 0,C 180,E1 4555.988,E2 4555.988} C_VEL
LIN {X 0,Y 102.896,Z 793.646,A -85,B 0,C 180,E1 4544.819,E2 4544.819} C_VEL
LIN {X 0,Y 114.323,Z 785.031,A -85,B 0,C 180,E1 4535.575,E2 4535.575} C_VEL
LIN {X 0,Y 127.475,Z 774.798,A -85,B 0,C 180,E1 4528.543,E2 4528.543} C_VEL
LIN {X 0,Y 141.412,Z 762.986,A -85,B 0,C 180,E1 4523.198,E2 4523.198} C_VEL
LIN {X 0,Y 155.665,Z 749.525,A -85,B 0,C 180,E1 4519.121,E2 4519.121} C_VEL
LIN {X 0,Y 168.843,Z 735.44,A -85,B 0,C 180,E1 4516.16,E2 4516.16} C_VEL
LIN {X 0,Y 181.722,Z 719.65,A -85,B 0,C 180,E1 4513.809,E2 4513.809} C_VEL
LIN {X 0,Y 193.747,Z 702.505,A -85,B 0,C 180,E1 4512,E2 4512} C_VEL
LIN {X 0,Y 204.486,Z 684.384,A -85,B 0,C 180,E1 4510.646,E2 4510.646} C_VEL
LIN {X 0,Y 213.978,Z 664.99,A -85,B 0,C 180,E1 4509.628,E2 4509.628} C_VEL
LIN {X 0,Y 221.617,Z 645.415,A -85,B 0,C 180,E1 4508.877,E2 4508.877} C_VEL
LIN {X 0,Y 227.701,Z 624.684,A -85,B 0,C 180,E1 4508.264,E2 4508.264} C_VEL
LIN {X 0,Y 231.906,Z 603.656,A -85,B 0,C 180,E1 4507.776,E2 4507.776} C_VEL
LIN {X 0,Y 241.705,Z 519.132,A -85,B 0,C 180,E1 4506.239,E2 4506.239} C_VEL
LIN {X 0,Y 240.66,Z 515.225,A -85,B 0,C 180,E1 4503.692,E2 4503.692} C_VEL
LIN {X 0,Y 240.023,Z 512.685,A -85,B 0,C 180,E1 4501.432,E2 4501.432} C_VEL
LIN {X 0,Y 239.616,Z 510.589,A -85,B 0,C 180,E1 4498.565,E2 4498.565} C_VEL
LIN {X 0,Y 239.776,Z 510.326,A -85,B 0,C 180,E1 4494.256,E2 4494.256} C_VEL
LIN {X 0,Y 240.297,Z 511.038,A -85,B 0,C 180,E1 4492.002,E2 4492.002} C_VEL
LIN {X 0,Y 241.622,Z 514.446,A -85,B 0,C 180,E1 4488.422,E2 4488.422} C_VEL
LIN {X 0,Y 241.932,Z 515.521,A -85,B 0,C 180,E1 4487.738,E2 4487.738} C_VEL
LIN {X 0,Y 234.06,Z 586.707,A -85,B 0,C 180,E1 4486.406,E2 4486.406} C_VEL
LIN {X 0,Y 231.001,Z 606.336,A -85,B 0,C 180,E1 4485.82,E2 4485.82} C_VEL
LIN {X 0,Y 226.379,Z 625.497,A -85,B 0,C 180,E1 4485.047,E2 4485.047} C_VEL
LIN {X 0,Y 220.41,Z 643.634,A -85,B 0,C 180,E1 4484.087,E2 4484.087} C_VEL
LIN {X 0,Y 212.472,Z 662.413,A -85,B 0,C 180,E1 4482.796,E2 4482.796} C_VEL
LIN {X 0,Y 203.269,Z 679.933,A -85,B 0,C 180,E1 4481.238,E2 4481.238} C_VEL
LIN {X 0,Y 192.929,Z 696.248,A -85,B 0,C 180,E1 4479.338,E2 4479.338} C_VEL
LIN {X 0,Y 181.209,Z 711.831,A -85,B 0,C 180,E1 4476.935,E2 4476.935} C_VEL
LIN {X 0,Y 168.67,Z 726.01,A -85,B 0,C 180,E1 4473.981,E2 4473.981} C_VEL
LIN {X 0,Y 155.439,Z 738.839,A -85,B 0,C 180,E1 4470.269,E2 4470.269} C_VEL
LIN {X 0,Y 142.568,Z 749.651,A -85,B 0,C 180,E1 4465.846,E2 4465.846} C_VEL
LIN {X 0,Y 129.813,Z 759.013,A -85,B 0,C 180,E1 4460.26,E2 4460.26} C_VEL
LIN {X 0,Y 117.984,Z 766.672,A -85,B 0,C 180,E1 4453.347,E2 4453.347} C_VEL
LIN {X 0,Y 107.423,Z 772.79,A -85,B 0,C 180,E1 4444.594,E2 4444.594} C_VEL
LIN {X 0,Y 99.483,Z 777.018,A -85,B 0,C 180,E1 4434.334,E2 4434.334} C_VEL
LIN {X 0,Y 94.558,Z 779.51,A -85,B 0,C 180,E1 4422.829,E2 4422.829} C_VEL
LIN {X 0,Y 92.84,Z 780.375,A -85,B 0,C 180,E1 4410.617,E2 4410.617} C_VEL
LIN {X 0,Y 94.075,Z 779.741,A -85,B 0,C 180,E1 4398.971,E2 4398.971} C_VEL
LIN {X 0,Y 98.502,Z 777.524,A -85,B 0,C 180,E1 4387.312,E2 4387.312} C_VEL
LIN {X 0,Y 105.995,Z 773.595,A -85,B 0,C 180,E1 4376.832,E2 4376.832} C_VEL
LIN {X 0,Y 115.617,Z 768.141,A -85,B 0,C 180,E1 4368.251,E2 4368.251} C_VEL
LIN {X 0,Y 127.201,Z 760.858,A -85,B 0,C 180,E1 4361.011,E2 4361.011} C_VEL
LIN {X 0,Y 139.58,Z 752.061,A -85,B 0,C 180,E1 4355.255,E2 4355.255} C_VEL
LIN {X 0,Y 152.261,Z 741.791,A -85,B 0,C 180,E1 4350.659,E2 4350.659} C_VEL
LIN {X 0,Y 164.867,Z 730.079,A -85,B 0,C 180,E1 4346.941,E2 4346.941} C_VEL
LIN {X 0,Y 177.156,Z 716.89,A -85,B 0,C 180,E1 4343.894,E2 4343.894} C_VEL
LIN {X 0,Y 188.428,Z 702.85,A -85,B 0,C 180,E1 4341.478,E2 4341.478} C_VEL
LIN {X 0,Y 198.855,Z 687.656,A -85,B 0,C 180,E1 4339.484,E2 4339.484} C_VEL
LIN {X 0,Y 208.453,Z 671.011,A -85,B 0,C 180,E1 4337.808,E2 4337.808} C_VEL
LIN {X 0,Y 216.817,Z 653.35,A -85,B 0,C 180,E1 4336.429,E2 4336.429} C_VEL
LIN {X 0,Y 223.891,Z 634.523,A -85,B 0,C 180,E1 4335.293,E2 4335.293} C_VEL
LIN {X 0,Y 229.505,Z 614.573,A -85,B 0,C 180,E1 4334.379,E2 4334.379} C_VEL
LIN {X 0,Y 233.386,Z 594.183,A -85,B 0,C 180,E1 4333.688,E2 4333.688} C_VEL
LIN {X 0,Y 238.385,Z 550.093,A -85,B 0,C 180,E1 4332.75,E2 4332.75} C_VEL
LIN {X 0,Y 242.226,Z 515.518,A -85,B 0,C 180,E1 4332.153,E2 4332.153} C_VEL
LIN {X 0,Y 241.163,Z 512.939,A -85,B 0,C 180,E1 4329.787,E2 4329.787} C_VEL
LIN {X 0,Y 240.324,Z 510.761,A -85,B 0,C 180,E1 4326.93,E2 4326.93} C_VEL
LIN {X 0,Y 239.857,Z 510.626,A -85,B 0,C 180,E1 4322.39,E2 4322.39} C_VEL
LIN {X 0,Y 239.975,Z 511.274,A -85,B 0,C 180,E1 4320.667,E2 4320.667} C_VEL
LIN {X 0,Y 240.597,Z 514.157,A -85,B 0,C 180,E1 4317.38,E2 4317.38} C_VEL
LIN {X 0,Y 241.615,Z 517.981,A -85,B 0,C 180,E1 4314.539,E2 4314.539} C_VEL
LIN {X 0,Y 241.929,Z 519.643,A -85,B 0,C 180,E1 4313.751,E2 4313.751} C_VEL
LIN {X 0,Y 231.976,Z 604.943,A -85,B 0,C 180,E1 4312.211,E2 4312.211} C_VEL
LIN {X 0,Y 227.648,Z 625.941,A -85,B 0,C 180,E1 4311.718,E2 4311.718} C_VEL
LIN {X 0,Y 221.622,Z 646.151,A -85,B 0,C 180,E1 4311.115,E2 4311.115} C_VEL
LIN {X 0,Y 213.982,Z 665.58,A -85,B 0,C 180,E1 4310.365,E2 4310.365} C_VEL
LIN {X 0,Y 204.49,Z 684.835,A -85,B 0,C 180,E1 4309.346,E2 4309.346} C_VEL
LIN {X 0,Y 193.865,Z 702.702,A -85,B 0,C 180,E1 4308.007,E2 4308.007} C_VEL
LIN {X 0,Y 182.183,Z 719.358,A -85,B 0,C 180,E1 4306.259,E2 4306.259} C_VEL
LIN {X 0,Y 168.917,Z 735.615,A -85,B 0,C 180,E1 4303.848,E2 4303.848} C_VEL
LIN {X 0,Y 155.583,Z 749.831,A -85,B 0,C 180,E1 4300.851,E2 4300.851} C_VEL
LIN {X 0,Y 141.417,Z 763.16,A -85,B 0,C 180,E1 4296.796,E2 4296.796} C_VEL
LIN {X 0,Y 127.309,Z 775.078,A -85,B 0,C 180,E1 4291.376,E2 4291.376} C_VEL
LIN {X 0,Y 125.033,Z 776.84,A -85,B 0,C 180,E1 4290.328,E2 4290.328} C_VEL
LIN {X 0,Y 119.644,Z 780.505,A -85,B 0,C 180,E1 4288.303,E2 4288.303} C_VEL
LIN {X 0,Y 103.917,Z 788.435,A -85,B 0,C 180,E1 4283.293,E2 4283.293} C_VEL
LIN {X 0,Y 98.999,Z 791.173,A -85,B 0,C 180,E1 4280.308,E2 4280.308} C_VEL
LIN {X 0,Y 89.495,Z 797.808,A -85,B 0,C 180,E1 4269.554,E2 4269.554} C_VEL
LIN {X 0,Y 83.509,Z 802.905,A -85,B 0,C 180,E1 4256.109,E2 4256.109} C_VEL
LIN {X 0,Y 82.208,Z 806.044,A -85,B 0,C 180,E1 4241.932,E2 4241.932} C_VEL
LIN {X 0,Y 83.991,Z 807.245,A -85,B 0,C 180,E1 4230.588,E2 4230.588} C_VEL
LIN {X 0,Y 83.384,Z 807.03,A -85,B 0,C 180,E1 4226.563,E2 4226.563} C_VEL
LIN {X 0,Y 82.141,Z 805.282,A -85,B 0,C 180,E1 4213.742,E2 4213.742} C_VEL
LIN {X 0,Y 84.867,Z 801.532,A -85,B 0,C 180,E1 4199.563,E2 4199.563} C_VEL
LIN {X 0,Y 92.102,Z 795.911,A -85,B 0,C 180,E1 4186.85,E2 4186.85} C_VEL
LIN {X 0,Y 103.09,Z 788.327,A -85,B 0,C 180,E1 4176.391,E2 4176.391} C_VEL
LIN {X 0,Y 116.107,Z 779.176,A -85,B 0,C 180,E1 4168.556,E2 4168.556} C_VEL
LIN {X 0,Y 130.823,Z 767.94,A -85,B 0,C 180,E1 4162.465,E2 4162.465} C_VEL
LIN {X 0,Y 145.187,Z 755.703,A -85,B 0,C 180,E1 4158.133,E2 4158.133} C_VEL
LIN {X 0,Y 159.305,Z 742.07,A -85,B 0,C 180,E1 4154.865,E2 4154.865} C_VEL
LIN {X 0,Y 173.069,Z 726.822,A -85,B 0,C 180,E1 4152.342,E2 4152.342} C_VEL
LIN {X 0,Y 186.032,Z 710.124,A -85,B 0,C 180,E1 4150.411,E2 4150.411} C_VEL
LIN {X 0,Y 197.404,Z 692.878,A -85,B 0,C 180,E1 4149.012,E2 4149.012} C_VEL
LIN {X 0,Y 207.467,Z 674.649,A -85,B 0,C 180,E1 4147.965,E2 4147.965} C_VEL
LIN {X 0,Y 216.181,Z 655.296,A -85,B 0,C 180,E1 4147.173,E2 4147.173} C_VEL
LIN {X 0,Y 223.171,Z 635.374,A -85,B 0,C 180,E1 4146.555,E2 4146.555} C_VEL
LIN {X 0,Y 228.427,Z 614.833,A -85,B 0,C 180,E1 4146.053,E2 4146.053} C_VEL
LIN {X 0,Y 231.864,Z 593.892,A -85,B 0,C 180,E1 4145.639,E2 4145.639} C_VEL
LIN {X 0,Y 239.884,Z 524.505,A -85,B 0,C 180,E1 4144.422,E2 4144.422} C_VEL
LIN {X 0,Y 238.911,Z 520.38,A -85,B 0,C 180,E1 4140.959,E2 4140.959} C_VEL
LIN {X 0,Y 238.604,Z 518.485,A -85,B 0,C 180,E1 4138.319,E2 4138.319} C_VEL
LIN {X 0,Y 238.836,Z 518.302,A -85,B 0,C 180,E1 4133.992,E2 4133.992} C_VEL
LIN {X 0,Y 239.254,Z 518.975,A -85,B 0,C 180,E1 4132.193,E2 4132.193} C_VEL
LIN {X 0,Y 240.118,Z 521.439,A -85,B 0,C 180,E1 4129.523,E2 4129.523} C_VEL
LIN {X 0,Y 232.606,Z 587.716,A -85,B 0,C 180,E1 4128.324,E2 4128.324} C_VEL
LIN {X 0,Y 229.46,Z 607.309,A -85,B 0,C 180,E1 4127.759,E2 4127.759} C_VEL
LIN {X 0,Y 224.707,Z 626.53,A -85,B 0,C 180,E1 4127.017,E2 4127.017} C_VEL
LIN {X 0,Y 218.386,Z 645.241,A -85,B 0,C 180,E1 4126.071,E2 4126.071} C_VEL
LIN {X 0,Y 210.187,Z 664.05,A -85,B 0,C 180,E1 4124.832,E2 4124.832} C_VEL
LIN {X 0,Y 200.873,Z 681.311,A -85,B 0,C 180,E1 4123.367,E2 4123.367} C_VEL
LIN {X 0,Y 190.245,Z 697.637,A -85,B 0,C 180,E1 4121.553,E2 4121.553} C_VEL
LIN {X 0,Y 178.045,Z 713.365,A -85,B 0,C 180,E1 4119.228,E2 4119.228} C_VEL
LIN {X 0,Y 165.69,Z 726.92,A -85,B 0,C 180,E1 4116.523,E2 4116.523} C_VEL
LIN {X 0,Y 152.473,Z 739.373,A -85,B 0,C 180,E1 4113.097,E2 4113.097} C_VEL
LIN {X 0,Y 138.83,Z 750.45,A -85,B 0,C 180,E1 4108.764,E2 4108.764} C_VEL
LIN {X 0,Y 125.006,Z 760.153,A -85,B 0,C 180,E1 4103.113,E2 4103.113} C_VEL
LIN {X 0,Y 112.346,Z 767.883,A -85,B 0,C 180,E1 4096.126,E2 4096.126} C_VEL
LIN {X 0,Y 100.993,Z 773.997,A -85,B 0,C 180,E1 4087.15,E2 4087.15} C_VEL
LIN {X 0,Y 92.317,Z 778.223,A -85,B 0,C 180,E1 4076.362,E2 4076.362} C_VEL
LIN {X 0,Y 86.856,Z 780.714,A -85,B 0,C 180,E1 4063.989,E2 4063.989} C_VEL
LIN {X 0,Y 84.931,Z 781.576,A -85,B 0,C 180,E1 4050.675,E2 4050.675} C_VEL
LIN {X 0,Y 86.318,Z 780.943,A -85,B 0,C 180,E1 4037.966,E2 4037.966} C_VEL
LIN {X 0,Y 91.239,Z 778.726,A -85,B 0,C 180,E1 4025.392,E2 4025.392} C_VEL
LIN {X 0,Y 99.448,Z 774.799,A -85,B 0,C 180,E1 4014.33,E2 4014.33} C_VEL
LIN {X 0,Y 109.825,Z 769.346,A -85,B 0,C 180,E1 4005.493,E2 4005.493} C_VEL
LIN {X 0,Y 122.142,Z 762.067,A -85,B 0,C 180,E1 3998.202,E2 3998.202} C_VEL
LIN {X 0,Y 135.159,Z 753.275,A -85,B 0,C 180,E1 3992.509,E2 3992.509} C_VEL
LIN {X 0,Y 149.179,Z 742.345,A -85,B 0,C 180,E1 3987.787,E2 3987.787} C_VEL
LIN {X 0,Y 162.268,Z 730.507,A -85,B 0,C 180,E1 3984.229,E2 3984.229} C_VEL
LIN {X 0,Y 174.96,Z 717.175,A -85,B 0,C 180,E1 3981.333,E2 3981.333} C_VEL
LIN {X 0,Y 186.668,Z 702.82,A -85,B 0,C 180,E1 3979.026,E2 3979.026} C_VEL
LIN {X 0,Y 197.251,Z 687.577,A -85,B 0,C 180,E1 3977.163,E2 3977.163} C_VEL
LIN {X 0,Y 206.628,Z 671.559,A -85,B 0,C 180,E1 3975.652,E2 3975.652} C_VEL
LIN {X 0,Y 215.174,Z 653.799,A -85,B 0,C 180,E1 3974.346,E2 3974.346} C_VEL
LIN {X 0,Y 222.239,Z 635.333,A -85,B 0,C 180,E1 3973.293,E2 3973.293} C_VEL
LIN {X 0,Y 227.976,Z 615.339,A -85,B 0,C 180,E1 3972.421,E2 3972.421} C_VEL
LIN {X 0,Y 231.933,Z 595.031,A -85,B 0,C 180,E1 3971.761,E2 3971.761} C_VEL
LIN {X 0,Y 237.087,Z 550.755,A -85,B 0,C 180,E1 3970.853,E2 3970.853} C_VEL
LIN {X 0,Y 240.401,Z 521.512,A -85,B 0,C 180,E1 3970.363,E2 3970.363} C_VEL
LIN {X 0,Y 239.297,Z 518.666,A -85,B 0,C 180,E1 3966.719,E2 3966.719} C_VEL
LIN {X 0,Y 238.877,Z 518.617,A -85,B 0,C 180,E1 3962.159,E2 3962.159} C_VEL
LIN {X 0,Y 238.985,Z 519.502,A -85,B 0,C 180,E1 3960.48,E2 3960.48} C_VEL
LIN {X 0,Y 239.478,Z 521.981,A -85,B 0,C 180,E1 3957.727,E2 3957.727} C_VEL
LIN {X 0,Y 240.149,Z 524.875,A -85,B 0,C 180,E1 3955.546,E2 3955.546} C_VEL
LIN {X 0,Y 230.682,Z 604.257,A -85,B 0,C 180,E1 3954.178,E2 3954.178} C_VEL
LIN {X 0,Y 226.318,Z 625.089,A -85,B 0,C 180,E1 3953.723,E2 3953.723} C_VEL
LIN {X 0,Y 220.273,Z 645.123,A -85,B 0,C 180,E1 3953.176,E2 3953.176} C_VEL
LIN {X 0,Y 212.775,Z 664.027,A -85,B 0,C 180,E1 3952.519,E2 3952.519} C_VEL
LIN {X 0,Y 203.143,Z 683.398,A -85,B 0,C 180,E1 3951.603,E2 3951.603} C_VEL
LIN {X 0,Y 192.175,Z 701.559,A -85,B 0,C 180,E1 3950.371,E2 3950.371} C_VEL
LIN {X 0,Y 179.943,Z 718.616,A -85,B 0,C 180,E1 3948.725,E2 3948.725} C_VEL
LIN {X 0,Y 166.558,Z 734.579,A -85,B 0,C 180,E1 3946.523,E2 3946.523} C_VEL
LIN {X 0,Y 152.184,Z 749.379,A -85,B 0,C 180,E1 3943.576,E2 3943.576} C_VEL
LIN {X 0,Y 137.513,Z 762.58,A -85,B 0,C 180,E1 3939.707,E2 3939.707} C_VEL
LIN {X 0,Y 122.935,Z 774.245,A -85,B 0,C 180,E1 3934.523,E2 3934.523} C_VEL
LIN {X 0,Y 108.994,Z 784.336,A -85,B 0,C 180,E1 3927.558,E2 3927.558} C_VEL
LIN {X 0,Y 98.999,Z 791.173,A -85,B 0,C 180,E1 3920.308,E2 3920.308} C_VEL
LIN {X 0,Y 94.331,Z 793.782,A -85,B 0,C 180,E1 3916.965,E2 3916.965} C_VEL
LIN {X 0,Y 80.87,Z 798.949,A -85,B 0,C 180,E1 3907.72,E2 3907.72} C_VEL
LIN {X 0,Y 77.511,Z 800.568,A -85,B 0,C 180,E1 3902.778,E2 3902.778} C_VEL
LIN {X 0,Y 74.215,Z 804.27,A -85,B 0,C 180,E1 3886.959,E2 3886.959} C_VEL
LIN {X 0,Y 75.459,Z 805.862,A -85,B 0,C 180,E1 3873.038,E2 3873.038} C_VEL
LIN {X 0,Y 75.99,Z 806.028,A -85,B 0,C 180,E1 3869.467,E2 3869.467} C_VEL
LIN {X 0,Y 74.209,Z 804.782,A -85,B 0,C 180,E1 3856.759,E2 3856.759} C_VEL
LIN {X 0,Y 76.212,Z 801.556,A -85,B 0,C 180,E1 3840.961,E2 3840.961} C_VEL
LIN {X 0,Y 83.236,Z 796.479,A -85,B 0,C 180,E1 3826.789,E2 3826.789} C_VEL
LIN {X 0,Y 94.398,Z 789.488,A -85,B 0,C 180,E1 3815.358,E2 3815.358} C_VEL
LIN {X 0,Y 107.739,Z 780.951,A -85,B 0,C 180,E1 3807.014,E2 3807.014} C_VEL
LIN {X 0,Y 122.056,Z 770.983,A -85,B 0,C 180,E1 3800.958,E2 3800.958} C_VEL
LIN {X 0,Y 136.611,Z 759.652,A -85,B 0,C 180,E1 3796.511,E2 3796.511} C_VEL
LIN {X 0,Y 150.961,Z 747,A -85,B 0,C 180,E1 3793.195,E2 3793.195} C_VEL
LIN {X 0,Y 165.296,Z 732.474,A -85,B 0,C 180,E1 3790.605,E2 3790.605} C_VEL
LIN {X 0,Y 178.339,Z 717.175,A -85,B 0,C 180,E1 3788.706,E2 3788.706} C_VEL
LIN {X 0,Y 190.774,Z 700.081,A -85,B 0,C 180,E1 3787.225,E2 3787.225} C_VEL
LIN {X 0,Y 201.627,Z 682.331,A -85,B 0,C 180,E1 3786.151,E2 3786.151} C_VEL
LIN {X 0,Y 211.381,Z 662.929,A -85,B 0,C 180,E1 3785.337,E2 3785.337} C_VEL
LIN {X 0,Y 219.258,Z 643.157,A -85,B 0,C 180,E1 3784.725,E2 3784.725} C_VEL
LIN {X 0,Y 225.387,Z 622.689,A -85,B 0,C 180,E1 3784.227,E2 3784.227} C_VEL
LIN {X 0,Y 229.672,Z 601.778,A -85,B 0,C 180,E1 3783.811,E2 3783.811} C_VEL
LIN {X 0,Y 238.268,Z 530.43,A -85,B 0,C 180,E1 3782.645,E2 3782.645} C_VEL
LIN {X 0,Y 237.776,Z 527.887,A -85,B 0,C 180,E1 3780.24,E2 3780.24} C_VEL
LIN {X 0,Y 237.596,Z 526.381,A -85,B 0,C 180,E1 3778.07,E2 3778.07} C_VEL
LIN {X 0,Y 237.865,Z 526.25,A -85,B 0,C 180,E1 3773.967,E2 3773.967} C_VEL
LIN {X 0,Y 238.211,Z 526.899,A -85,B 0,C 180,E1 3772.402,E2 3772.402} C_VEL
LIN {X 0,Y 238.456,Z 528.071,A -85,B 0,C 180,E1 3771.324,E2 3771.324} C_VEL
LIN {X 0,Y 231.322,Z 589.425,A -85,B 0,C 180,E1 3770.247,E2 3770.247} C_VEL
LIN {X 0,Y 228.042,Z 608.919,A -85,B 0,C 180,E1 3769.701,E2 3769.701} C_VEL
LIN {X 0,Y 223.305,Z 627.563,A -85,B 0,C 180,E1 3769.015,E2 3769.015} C_VEL
LIN {X 0,Y 217.088,Z 645.659,A -85,B 0,C 180,E1 3768.153,E2 3768.153} C_VEL
LIN {X 0,Y 208.731,Z 664.585,A -85,B 0,C 180,E1 3766.988,E2 3766.988} C_VEL
LIN {X 0,Y 198.839,Z 682.549,A -85,B 0,C 180,E1 3765.556,E2 3765.556} C_VEL
LIN {X 0,Y 187.897,Z 698.953,A -85,B 0,C 180,E1 3763.836,E2 3763.836} C_VEL
LIN {X 0,Y 175.842,Z 714.135,A -85,B 0,C 180,E1 3761.724,E2 3761.724} C_VEL
LIN {X 0,Y 162.701,Z 728.173,A -85,B 0,C 180,E1 3759.079,E2 3759.079} C_VEL
LIN {X 0,Y 149.063,Z 740.606,A -85,B 0,C 180,E1 3755.812,E2 3755.812} C_VEL
LIN {X 0,Y 135.111,Z 751.51,A -85,B 0,C 180,E1 3751.716,E2 3751.716} C_VEL
LIN {X 0,Y 120.926,Z 761.042,A -85,B 0,C 180,E1 3746.358,E2 3746.358} C_VEL
LIN {X 0,Y 107.001,Z 769.093,A -85,B 0,C 180,E1 3739.19,E2 3739.19} C_VEL
